    60:(* get P171 index 0 *)
        fbTD20Transaction.i_wPKE := 16#6000 OR 171;
        fbTD20Transaction.i_bIND := 0;
        fbTD20Transaction.i_dwPWE := 0;
        fbTD20Transaction.i_xExecute := TRUE;
        IF fbTD20Transaction.q_xError THEN
            iCatch := iCatch +1;
            a_TransactionErrorMesg();
            iStep := 9000;
        ELSIF fbTD20Transaction.q_xDone THEN
            fbTD20Transaction.i_xExecute := FALSE;
            IF fbTD20Transaction.q_wPKE = (16#4000 OR 171) THEN
                q_stStatus.wErrorCode_P171 := DWORD_TO_WORD(fbTD20Transaction.q_dwPWE);
                iStep := 8000;
            ELSE
                a_DriverErrorMesg();
                iStep := 9100;
            END_IF
        END_IF

    8000: (* done *)
        q_xDone := TRUE;
        IF  i_xExecute = FALSE THEN
            q_xDone:= FALSE;
            iStep := 0;
        END_IF

    9000: (* Transaction Error *)
        q_xError := TRUE;

    9100: (* Driver Error *)
        q_xError := TRUE;

END_CASE

fbTD20Transaction(
    i_wControlWord:= i_wControlWord,
    i_tTimeOut:= i_tTimeOut,
    iq_stSerialRXBuffer:= iq_stSerialRXBuffer,
    iq_stSerialTXBuffer:= iq_stSerialTXBuffer,
    q_wStatusWord=> q_stStatus.wStatusWord,
    q_wFrequency_P3=>  q_stStatus.wFrequency_P3,
    q_wVoltage_P4=> q_stStatus.wVoltage_P4,
    q_wMotorCurrent_P5=> q_stStatus.wMotorCurrent_P5,
    q_wConverterTemp_P11=> q_stStatus.wConverterTemp_P11,
    q_wPumpTemp_P127=> q_stStatus.wPumpTemp_P127);

IF fbTD20Transaction.q_xError THEN
    a_ClearStatus();
END_IF

q_abLastSentArray := fbTD20Transaction.q_abLastSentArray;
q_abLastReceivedArray := fbTD20Transaction.q_abLastReceivedArray;

ACTION a_ClearStatus:
q_stStatus.wStatusWord := 0;
q_stStatus.wFrequency_P3 := 0;
q_stStatus.wVoltage_P4 := 0;
q_stStatus.wMotorCurrent_P5 := 0;
q_stStatus.wConverterTemp_P11 := 0;
q_stStatus.wCriticalFreq_P20 := 0;
q_stStatus.wMaxCurrentFactor_P21 := 0;
q_stStatus.wSetpointFreq_P24 := 0;
q_stStatus.wMaxRunUpTime_P32 := 0;
q_stStatus.wPumpTemp_P127 := 0;
q_stStatus.wErrorCode_P171 := 0;
END_ACTION

ACTION a_DriverErrorMesg:
fbFormatString( sformat:=sDriverErrMesg,
    arg1:=F_INT(iStep),
    arg2:=F_WORD(fbTD20Transaction.q_wPKE),
    sOut => q_sResult);

a_ClearStatus();
END_ACTION

ACTION a_TransactionErrorMesg:
fbFormatString( sformat:=sTransactionErrMesg,
    arg1:=F_INT(iStep),
    arg2:=F_STRING(fbTD20Transaction.q_sResult),
    sOut => q_sResult);

a_ClearStatus();
q_xTimeout := fbTD20Transaction.q_xTimeout;
END_ACTION

END_FUNCTION_BLOCK

// ---- POUs/Serial drivers/Pumps/Oerlikon TD20/FB_TD20Transaction.TcPOU
FUNCTION_BLOCK FB_TD20Transaction
VAR_INPUT
    /// rising edge execute
    i_xExecute: BOOL;
    /// RS-485 Addrress of Pump, 0 if RS-232
    i_bAddress: BYTE;
    /// PKE Parameter number and type of access
    i_wPKE: WORD;
    /// IND Parameter index
    i_bIND: BYTE;
    /// PWE Parameter value
    i_dwPWE: DWORD;
    /// Control Word
    i_wControlWord: WORD;
    /// Maximum wait time for reply
    i_tTimeOut: TIME := TIME#1s0ms;
END_VAR
VAR_OUTPUT
    q_xDone: BOOL;
    q_xError: BOOL;
    q_xTimeout: BOOL;
    q_sResult: STRING(MAX_STRING_LENGTH);
    /// Sent data
    q_abSendData: ARRAY[0..23] OF BYTE;
    /// Received Data data
    q_abResponseData: ARRAY[0..23] OF BYTE;
    /// Received PKE
    q_wPKE: WORD;
    /// Received PWE
    q_dwPWE: DWORD;
    /// Received Status Word
    q_wStatusWord: WORD;
    /// Current stator frequency
    q_wFrequency_P3: WORD;
    /// Current intermediate circuit voltage
    q_wVoltage_P4: WORD;
    /// Current motor current
    q_wMotorCurrent_P5: WORD;
    /// Current frequency converter temperature
    q_wConverterTemp_P11: WORD;
    /// Current pump temperature
    q_wPumpTemp_P127: WORD;
    /// Last Byte Sequence Sent to Serial Device - for debugging
    q_abLastSentArray: ARRAY[0..23] OF BYTE;
    /// Last Byte Sequence Received from Serial Device - for debugging
    q_abLastReceivedArray: ARRAY[0..23] OF BYTE;
END_VAR
VAR_IN_OUT
    iq_stSerialRXBuffer: ComBuffer;
    iq_stSerialTXBuffer: ComBuffer;
END_VAR
VAR
    rtExecute: R_TRIG;
    iStep: INT;
    fbClearComBuffer: ClearComBuffer;
    tonTimeout: TON;
    wTemp: WORD;
    dwTemp: DWORD;
    i: INT;
    fbSendData: SendData;
    fbReceiveData: ReceiveData;
    bRXChecksum: BYTE;
    bRXAddress: BYTE;
    nPrefix : BYTE := 16#02;
END_VAR

(* This function block performs serial transactions with an Oerlikon TD20 *)

(* rising edge trigger *)
rtExecute(CLK:= i_xExecute);
IF rtExecute.Q THEN
    q_xDone	:= FALSE;
    q_xError := FALSE;
    q_xTimeout := FALSE;
    q_sResult:= '';
    MEMSET(destAddr:=ADR(q_abSendData), fillByte:=0, n:=SIZEOF(q_abSendData));
    MEMSET(destAddr:=ADR(q_abResponseData), fillByte:=0, n:=SIZEOF(q_abResponseData));
    iStep := 10;
END_IF

CASE iStep OF
    0:
        ; (* idle *)

    10: (* clear com buffers *)
        fbClearComBuffer(Buffer:= iq_stSerialRXBuffer);
        fbClearComBuffer(Buffer:= iq_stSerialTXBuffer);

        (* build the send data *)
        (* byte 0 STX *)
        q_abSendData[0] := 2; (* STX *)

        (* byte 1 LGE - Length *)
        q_abSendData[1] := 22;

        (* byte 2 ADR - Address for RS-485, use 0 for RS-232 *)
        q_abSendData[2] := i_bAddress;

        (* bytes 3-4 PKE - Parameter Number and Type of Access *)
        wTemp :=  HOST_TO_BE16(i_wPKE);
        MEMCPY(destAddr:= ADR(q_abSendData[3]), srcAddr:=ADR(wTemp), n:=2);

        (* byte 5 is reserved *)
        (* byte 6 IND - Parameter index *)
        q_abSendData[6] := i_bIND;

        (* bytes 7-10 - Parameter Value *)
        dwTemp := HOST_TO_BE32(i_dwPWE);
        MEMCPY(destAddr:= ADR(q_abSendData[7]), srcAddr:=ADR(dwTemp), n:=4);

        (* bytes 11-12 - control word *)
        wTemp :=  HOST_TO_BE16(i_wControlWord);
        MEMCPY(destAddr:= ADR(q_abSendData[11]), srcAddr:=ADR(wTemp), n:=2);

        (* rest of the bytes for any read or write are 0 *)
        (* generate checksum *)
        q_abSendData[23] := F_CalcTD20Checksum(i_abData:=q_abSendData);

        (* send the data *)
        fbSendData(
            pSendData:= ADR(q_abSendData),
            Length:= 24,
            TXbuffer:= iq_stSerialTXBuffer);


        q_abLastSentArray := q_abSendData;
        iStep := iStep + 10;

    20: (* Finish sending the data *)
        IF fbSendData.Busy THEN
            fbSendData( TXbuffer:= iq_stSerialTXBuffer );
        ELSIF fbSendData.Error <> 0 THEN
            q_sResult := CONCAT('In step 20 fbSendData resulted in error: ', INT_TO_STRING(fbSendData.Error));
            iStep := 9000;
        ELSIF NOT fbSendData.Busy THEN
            iStep := iStep + 10;
        END_IF
        (* Reset receive *)
        fbReceiveData(
            pReceiveData:= ADR(q_abResponseData),
            Reset:= TRUE,
            RXbuffer:= iq_stSerialRXBuffer);
        tonTimeout(IN:= FALSE);

    30: (* Get reply *)
        fbReceiveData(
            pReceiveData:= ADR(q_abResponseData),
            SizeReceiveData:= 24,
            Timeout:= i_tTimeOut,
            Reset:= FALSE,
            RXbuffer:= iq_stSerialRXBuffer,
            pPrefix := ADR(nPrefix), LenPrefix:=1 );
        tonTimeout(IN:= TRUE, PT:= i_tTimeOut);
        IF fbReceiveData.Error <> 0 THEN
            q_sResult := CONCAT('In step 30 fbReceiveData resulted in error: ', INT_TO_STRING(fbReceiveData.Error));
            iStep := 9000;
        ELSIF fbReceiveData.RxTimeout OR tonTimeout.Q THEN
            q_sResult := 'Device failed to reply within timeout period';
            q_xTimeout := TRUE;
            iStep := 9000;
        ELSIF fbReceiveData.DataReceived THEN
            q_abLastReceivedArray := q_abResponseData;
            bRXChecksum := F_CalcTD20Checksum(q_abResponseData);
            bRXAddress := q_abResponseData[2];
            MEMCPY(destAddr:=ADR(wTemp) , srcAddr:=ADR(q_abResponseData[3]), n:=2);
            q_wPKE := BE16_TO_HOST(wTemp);
            MEMCPY(destAddr:=ADR(dwTemp) , srcAddr:=ADR(q_abResponseData[7]), n:=4);
            q_dwPWE := BE32_TO_HOST(dwTemp);

            IF bRXChecksum <> q_abResponseData[23] THEN
                q_sResult := 'Invalid checksum on received data.';
                iStep := 9000;
            ELSIF i_bAddress <> bRXAddress THEN
                q_sResult := 'Invalid unit address on received data.';
                iStep := 9000;
            ELSIF (q_wPKE AND 16#F000) = 2#0111000000000000 THEN
                q_sResult := 'Frequency converter cannot run the command.';
                iStep := 9000;
            ELSIF (Q_wPKE AND 16#F000) = 2#1000000000000000 THEN
                q_sResult := 'During write access: no permission to write.';
                iStep := 9000;
            ELSE
                MEMCPY(destAddr:=ADR(wTemp) , srcAddr:=ADR(q_abResponseData[11]), n:=2);
                q_wStatusWord := BE16_TO_HOST(wTemp);
                MEMCPY(destAddr:=ADR(wTemp) , srcAddr:=ADR(q_abResponseData[13]), n:=2);
                q_wFrequency_P3:= BE16_TO_HOST(wTemp);
                MEMCPY(destAddr:=ADR(wTemp) , srcAddr:=ADR(q_abResponseData[21]), n:=2);
                q_wVoltage_P4:= BE16_TO_HOST(wTemp);
                MEMCPY(destAddr:=ADR(wTemp) , srcAddr:=ADR(q_abResponseData[17]), n:=2);
                q_wMotorCurrent_P5:= BE16_TO_HOST(wTemp);
                MEMCPY(destAddr:=ADR(wTemp) , srcAddr:=ADR(q_abResponseData[15]), n:=2);
                q_wConverterTemp_P11:= BE16_TO_HOST(wTemp);
                MEMCPY(destAddr:=ADR(wTemp) , srcAddr:=ADR(q_abResponseData[19]), n:=2);
                q_wPumpTemp_P127:= BE16_TO_HOST(wTemp);
                q_sResult := 'Success.';
                q_xDone:= TRUE;
                iStep := 100;
            END_IF
        END_IF

    100: (* done *)
        IF  i_xExecute = FALSE THEN
            q_xDone:= FALSE;
            iStep := 0;
        END_IF

    9000:
        q_wPKE:= 0;
        q_dwPWE:= 0;
        q_wStatusWord:= 0;
        q_wFrequency_P3:= 0;
        q_wVoltage_P4:= 0;
        q_wMotorCurrent_P5:= 0;
        q_wConverterTemp_P11:= 0;
        q_wPumpTemp_P127:= 0;
        q_xError := TRUE;;




END_CASE

END_FUNCTION_BLOCK

// ---- POUs/Serial drivers/Pumps/Oerlikon TD20/F_CalcTD20Checksum.TcPOU
FUNCTION F_CalcTD20Checksum : BYTE
VAR_INPUT
    i_abData: ARRAY[0..23] OF BYTE;
END_VAR
VAR
    bChecksum: BYTE;
    i: INT;
END_VAR

bChecksum := i_abData[0];
FOR i:=1 TO 22 DO
    bChecksum := bChecksum XOR i_abData[i];
END_FOR
F_CalcTD20Checksum := bChecksum;

END_FUNCTION

// ---- POUs/Serial drivers/Pumps/Oerlikon TD20/FB_OERLIKON_TO_PTM.TcPOU
FUNCTION_BLOCK FB_OERLIKON_TO_PTM
VAR_IN_OUT
    iq_stPTM: ST_LeyboldPTM;
    iq_stOerlikon_stat: ST_TD20Status;
END_VAR

(* This function block is used to map the IO points from the Oerlikon structures
to the generic turbo structures *)

(* Readbacks *)
iq_stPTM.i_xAccel := iq_stOerlikon_stat.wStatusWord.4;
iq_stPTM.i_xDecel := iq_stOerlikon_stat.wStatusWord.5;
iq_stPTM.i_xAtSpd := iq_stOerlikon_stat.wStatusWord.10;
iq_stPTM.q_xRemote := iq_stOerlikon_stat.wStatusWord.15; (* Remote control enabled *)
iq_stPTM.i_diCurSpd := WORD_TO_DINT(iq_stOerlikon_stat.wFrequency_P3);
iq_stPTM.i_diPwr := LREAL_TO_DINT(WORD_TO_DINT(iq_stOerlikon_stat.wMotorCurrent_P5 * iq_stOerlikon_stat.wVoltage_P4)*0.01); (*Current in units 0.1 A and voltage in units 0.1V, TD20 manual page 23*)
iq_stPTM.i_diElecTemp := WORD_TO_DINT(iq_stOerlikon_stat.wConverterTemp_P11);
//iq_stPTM.i_diPumpTemp := WORD_TO_DINT(iq_stOerlikon_stat.wPumpTemp_P127);

(* Faults and warnings *)
//iq_stPTM.xFault := iq_stOerlikon_stat.wStatusWord.3;
iq_stPTM.i_xTempFault := iq_stOerlikon_stat.wStatusWord.7; (* specified as a temperature warning but it could be a fault *)
//iq_stPTM.xWarn := iq_stOerlikon_stat.wStatusWord.14; (* warning summary bit *)

END_FUNCTION_BLOCK

// ---- POUs/Serial drivers/Pumps/Oerlikon TD400/FB_OERLIKON_TD400_COM.TcPOU
FUNCTION_BLOCK FB_OERLIKON_TD400_COM
VAR_INPUT
END_VAR
VAR
    tTimeOut : TIME := TIME#1S0MS;
    fbTD400SerialDriver : FB_TD400SerialDriver;
END_VAR
VAR_IN_OUT
    SerialRXBuffer : ComBuffer;
    SerialTXBuffer : ComBuffer;
    stTD400Control : ST_TD400Control;
END_VAR
VAR_OUTPUT
    stTD400Status : ST_TD400Status;
END_VAR

(* This program is called from Serial PTM IO *)

(* scan the pumps one at a time *)//MG???
fbTD400SerialDriver(
    i_xExecute:= TRUE,
    i_tTimeOut:= tTimeOut,
    i_wControlWord:= 16#0000,
    iq_stControl:= stTD400Control,
    iq_stSerialRXBuffer:= SerialRXBuffer,
    iq_stSerialTXBuffer:= SerialTXBuffer,
    q_xDone=> ,
    q_xError=> ,
    q_xTimeout=> ,
    q_sResult=> ,
    q_stStatus=> stTD400Status);

IF fbTD400SerialDriver.q_xDone
    OR fbTD400SerialDriver.q_xError
    OR fbTD400SerialDriver.q_xTimeout THEN
        (* reset for next time *)
        fbTD400SerialDriver(i_xExecute:= FALSE, iq_stSerialRXBuffer:= SerialRXBuffer, iq_stSerialTXBuffer:= SerialTXBuffer, iq_stControl:= stTD400Control);
END_IF

END_FUNCTION_BLOCK

// ---- POUs/Serial drivers/Pumps/Oerlikon TD400/FB_TD400SerialDriver.TcPOU
FUNCTION_BLOCK FB_TD400SerialDriver
VAR_INPUT
    /// rising edge execute
    i_xExecute: BOOL;
    /// Maximum wait time for reply
    i_tTimeOut: TIME := TIME#1s0ms;
    i_wControlWord: WORD;
END_VAR
VAR_OUTPUT
    q_xDone: BOOL;
    q_xError: BOOL;
    q_xTimeout: BOOL;
    q_sResult: STRING(255);
    q_stStatus: ST_TD400Status;
    /// Last Byte Sequence Sent to Serial Device - for debugging
    q_abLastSentArray: ARRAY[0..23] OF BYTE;
    /// Last Byte Sequence Received from Serial Device - for debugging
    q_abLastReceivedArray: ARRAY[0..23] OF BYTE;
END_VAR
VAR_IN_OUT
    iq_stSerialRXBuffer: ComBuffer;
    iq_stSerialTXBuffer: ComBuffer;
    iq_stControl: ST_TD400Control;
END_VAR
VAR
    rtExecute: R_TRIG;
    rtTransDone: R_TRIG;
    iStep: INT;
    fbTD400Transaction: FB_TD400Transaction;
    fbFormatString: FB_FormatString;
    iCatch: INT;
    sTransactionErrMesg : STRING := 'In step %d fbTD20Transaction failed with message: %s';
    sDriverErrMesg		: STRING := 'In step %d FB_TD20SerialDriver failed with unexpected PKE reply: %X';
    bSetFreq : BOOL := FALSE; //flag to write to controller to set new frequency
    nOldSetSetpointFreq_P24 : WORD; //local value for setpoint frequency parameter to compare with new value
    bControlDisabled : BOOL := TRUE; //flag to enable setting frequency
END_VAR

(* This function block performs serial transactions with a Oerlikon TD400 Pump controller *)
//Wait until all needed parameters received to enable control to set frequency
IF q_stStatus.wMinSetpointFreq_P19 <> 0 AND q_stStatus.wMaxSetpointFreq_P18 <> 0 AND q_stStatus.wSetpointFreq_P24 <> 0 THEN
    //On first pass update Set frequency parameter with value from controller
    IF bControlDisabled THEN
        iq_stControl.wSetSetpointFreq_P24 := q_stStatus.wSetpointFreq_P24;
        nOldSetSetpointFreq_P24 := q_stStatus.wSetpointFreq_P24;
        bControlDisabled := FALSE;
        bSetFreq := FALSE;
    ELSE
        IF nOldSetSetpointFreq_P24 <> iq_stControl.wSetSetpointFreq_P24 THEN
            nOldSetSetpointFreq_P24 := iq_stControl.wSetSetpointFreq_P24;
            bSetFreq := TRUE;
        END_IF
    END_IF
ELSE
    iq_stControl.wSetSetpointFreq_P24 := q_stStatus.wSetpointFreq_P24;
    bControlDisabled := TRUE;
    bSetFreq := FALSE;
END_IF

(* rising edge trigger *)
rtExecute(CLK:= i_xExecute);
IF rtExecute.Q  THEN
    q_xDone	:= FALSE;
    q_xError := FALSE;
    q_xTimeout := FALSE;
    q_sResult:= '';
    iStep := 10;
END_IF

CASE iStep OF
    0: (* idle *)
        ;

    10: (* assure rising edge *)
        fbTD400Transaction.i_xExecute := FALSE;
        iStep := iStep + 10;

    20:(* get P20 *)
        fbTD400Transaction.i_wPKE := 16#1000 OR 20;
        fbTD400Transaction.i_bIND := 0;
        fbTD400Transaction.i_dwPWE := 0;
        fbTD400Transaction.i_xExecute := TRUE;

        IF fbTD400Transaction.q_xError THEN
            iCatch := iCatch +1;
            a_TransactionErrorMesg();
            iStep := 9000;
        ELSIF fbTD400Transaction.q_xDone THEN
            fbTD400Transaction.i_xExecute := FALSE;
            IF fbTD400Transaction.q_wPKE = (16#1000 OR 20) THEN
                q_stStatus.wCriticalFreq_P20 := DWORD_TO_WORD(fbTD400Transaction.q_dwPWE);
                iStep := iStep + 10;
            ELSE
                a_DriverErrorMesg();
                iStep := 9100;
            END_IF
        END_IF

    30:(* set P24 *)
        IF bSetFreq THEN
            fbTD400Transaction.i_wPKE := 16#2000 OR 24;
            fbTD400Transaction.i_bIND := 0;
            fbTD400Transaction.i_dwPWE := WORD_TO_DWORD(iq_stControl.wSetSetpointFreq_P24);
            fbTD400Transaction.i_xExecute := TRUE;

            IF fbTD400Transaction.q_xError THEN
                iCatch := iCatch +1;
                a_TransactionErrorMesg();
                iStep := 9000;
                bSetFreq := FALSE;
            ELSIF fbTD400Transaction.q_xDone THEN
                fbTD400Transaction.i_xExecute := FALSE;
                bSetFreq := FALSE;
                IF fbTD400Transaction.q_wPKE = (16#1000 OR 24) THEN
                    q_stStatus.wSetpointFreq_P24 := DWORD_TO_WORD(fbTD400Transaction.q_dwPWE);
                    iStep := iStep + 10;
                ELSE
                    a_DriverErrorMesg();
                    iStep := 9100;
                END_IF
            END_IF
        ELSE
            iStep := iStep + 10;
        END_IF

    40:(* get P24 *)
        fbTD400Transaction.i_wPKE := 16#1000 OR 24;
        fbTD400Transaction.i_bIND := 0;
        fbTD400Transaction.i_dwPWE := 0;
        fbTD400Transaction.i_xExecute := TRUE;
        IF fbTD400Transaction.q_xError THEN
            iCatch := iCatch +1;
            a_TransactionErrorMesg();
            iStep := 9000;
        ELSIF fbTD400Transaction.q_xDone THEN
            fbTD400Transaction.i_xExecute := FALSE;
            IF fbTD400Transaction.q_wPKE = (16#1000 OR 24) THEN
                q_stStatus.wSetpointFreq_P24 := DWORD_TO_WORD(fbTD400Transaction.q_dwPWE);
                iStep := iStep + 10;
            ELSE
                a_DriverErrorMesg();
                iStep := 9100;
            END_IF
        END_IF

    50:(* get P32 *)
        fbTD400Transaction.i_wPKE := 16#1000 OR 32;
        fbTD400Transaction.i_bIND := 0;
        fbTD400Transaction.i_dwPWE := 0;
        fbTD400Transaction.i_xExecute := TRUE;
        IF fbTD400Transaction.q_xError THEN
            iCatch := iCatch +1;
            a_TransactionErrorMesg();
            iStep := 9000;
        ELSIF fbTD400Transaction.q_xDone THEN
            fbTD400Transaction.i_xExecute := FALSE;
            IF fbTD400Transaction.q_wPKE = (16#1000 OR 32) THEN
                q_stStatus.wMaxRunUpTime_P32 := DWORD_TO_WORD(fbTD400Transaction.q_dwPWE);
                iStep := iStep + 10;
            ELSE
                a_DriverErrorMesg();
                iStep := 9100;
            END_IF
        END_IF

    60:(* get P171 index 0 *)
        fbTD400Transaction.i_wPKE := 16#6000 OR 171;
        fbTD400Transaction.i_bIND := 0;
        fbTD400Transaction.i_dwPWE := 0;
        fbTD400Transaction.i_xExecute := TRUE;
        IF fbTD400Transaction.q_xError THEN
            iCatch := iCatch +1;
            a_TransactionErrorMesg();
            iStep := 9000;
        ELSIF fbTD400Transaction.q_xDone THEN
            fbTD400Transaction.i_xExecute := FALSE;
            IF fbTD400Transaction.q_wPKE = (16#4000 OR 171) THEN
                q_stStatus.wErrorCode_P171 := DWORD_TO_WORD(fbTD400Transaction.q_dwPWE);
                //iStep := 8000;
                iStep := iStep + 10;
            ELSE
                a_DriverErrorMesg();
                iStep := 9100;
            END_IF
        END_IF

    70:(* get P18 *)
        fbTD400Transaction.i_wPKE := 16#1000 OR 18;
        fbTD400Transaction.i_bIND := 0;
        fbTD400Transaction.i_dwPWE := 0;
        fbTD400Transaction.i_xExecute := TRUE;
        IF fbTD400Transaction.q_xError THEN
            iCatch := iCatch +1;
            a_TransactionErrorMesg();
            iStep := 9000;
        ELSIF fbTD400Transaction.q_xDone THEN
            fbTD400Transaction.i_xExecute := FALSE;
            IF fbTD400Transaction.q_wPKE = (16#1000 OR 18) THEN
                q_stStatus.wMaxSetpointFreq_P18 := DWORD_TO_WORD(fbTD400Transaction.q_dwPWE);
                iStep := iStep + 10;
            ELSE
                a_DriverErrorMesg();
                iStep := 9100;
            END_IF
        END_IF

    80:(* get P19 *)
        fbTD400Transaction.i_wPKE := 16#1000 OR 19;
        fbTD400Transaction.i_bIND := 0;
        fbTD400Transaction.i_dwPWE := 0;
        fbTD400Transaction.i_xExecute := TRUE;
        IF fbTD400Transaction.q_xError THEN
            iCatch := iCatch +1;
            a_TransactionErrorMesg();
            iStep := 9000;
        ELSIF fbTD400Transaction.q_xDone THEN
            fbTD400Transaction.i_xExecute := FALSE;
            IF fbTD400Transaction.q_wPKE = (16#1000 OR 19) THEN
                q_stStatus.wMinSetpointFreq_P19 := DWORD_TO_WORD(fbTD400Transaction.q_dwPWE);
                iStep := 8000;
            ELSE
                a_DriverErrorMesg();
                iStep := 9100;
            END_IF
        END_IF

    8000: (* done *)
        q_xDone := TRUE;
        IF  i_xExecute = FALSE THEN
            q_xDone:= FALSE;
            iStep := 0;
        END_IF

    9000: (* Transaction Error *)
        q_xError := TRUE;

    9100: (* Driver Error *)
        q_xError := TRUE;

END_CASE

fbTD400Transaction(
    i_wControlWord:= i_wControlWord,
    i_tTimeOut:= i_tTimeOut,
    iq_stSerialRXBuffer:= iq_stSerialRXBuffer,
    iq_stSerialTXBuffer:= iq_stSerialTXBuffer,
    q_wStatusWord=> q_stStatus.wStatusWord,
    q_wFrequency_P3=>  q_stStatus.wFrequency_P3,
    q_wVoltage_P4=> q_stStatus.wVoltage_P4,
    q_wMotorCurrent_P5=> q_stStatus.wMotorCurrent_P5,
    q_wConverterTemp_P11=> q_stStatus.wConverterTemp_P11,
    q_wPumpTemp_P127=> q_stStatus.wPumpTemp_P127);

IF fbTD400Transaction.q_xError THEN
    a_ClearStatus();
END_IF

q_abLastSentArray := fbTD400Transaction.q_abLastSentArray;
q_abLastReceivedArray := fbTD400Transaction.q_abLastReceivedArray;

ACTION a_ClearStatus:
q_stStatus.wStatusWord := 0;
q_stStatus.wFrequency_P3 := 0;
q_stStatus.wVoltage_P4 := 0;
q_stStatus.wMotorCurrent_P5 := 0;
q_stStatus.wConverterTemp_P11 := 0;
q_stStatus.wMaxSetpointFreq_P18 := 0;
q_stStatus.wMinSetpointFreq_P19 := 0;
q_stStatus.wCriticalFreq_P20 := 0;
//q_stStatus.wMaxCurrentFactor_P21 := 0;
q_stStatus.wSetpointFreq_P24 := 0;
q_stStatus.wMaxRunUpTime_P32 := 0;
q_stStatus.wPumpTemp_P127 := 0;
q_stStatus.wErrorCode_P171 := 0;
END_ACTION

ACTION a_DriverErrorMesg:
fbFormatString( sformat:=sDriverErrMesg,
    arg1:=F_INT(iStep),
    arg2:=F_WORD(fbTD400Transaction.q_wPKE),
    sOut => q_sResult);

a_ClearStatus();
END_ACTION

ACTION a_TransactionErrorMesg:
fbFormatString( sformat:=sTransactionErrMesg,
    arg1:=F_INT(iStep),
    arg2:=F_STRING(fbTD400Transaction.q_sResult),
    sOut => q_sResult);

a_ClearStatus();
q_xTimeout := fbTD400Transaction.q_xTimeout;
END_ACTION

END_FUNCTION_BLOCK

// ---- POUs/Serial drivers/Pumps/Oerlikon TD400/FB_TD400Transaction.TcPOU
FUNCTION_BLOCK FB_TD400Transaction
VAR_INPUT
    /// rising edge execute
    i_xExecute: BOOL;
    /// RS-485 Addrress of Pump, 0 if RS-232
    i_bAddress: BYTE;
    /// PKE Parameter number and type of access
    i_wPKE: WORD;
    /// IND Parameter index
    i_bIND: BYTE;
    /// PWE Parameter value
    i_dwPWE: DWORD;
    /// Control Word
    i_wControlWord: WORD;
    /// Maximum wait time for reply
    i_tTimeOut: TIME := TIME#1s0ms;
END_VAR
VAR_OUTPUT
    q_xDone: BOOL;
    q_xError: BOOL;
    q_xTimeout: BOOL;
    q_sResult: STRING(MAX_STRING_LENGTH);
    /// Sent data
    q_abSendData: ARRAY[0..23] OF BYTE;
    /// Received Data data
    q_abResponseData: ARRAY[0..23] OF BYTE;
    /// Received PKE
    q_wPKE: WORD;
    /// Received PWE
    q_dwPWE: DWORD;
    /// Received Status Word
    q_wStatusWord: WORD;
    /// Current stator frequency
    q_wFrequency_P3: WORD;
    /// Current intermediate circuit voltage
    q_wVoltage_P4: WORD;
    /// Current motor current
    q_wMotorCurrent_P5: WORD;
    /// Current frequency converter temperature
    q_wConverterTemp_P11: WORD;
    /// Current pump temperature
    q_wPumpTemp_P127: WORD;
    /// Last Byte Sequence Sent to Serial Device - for debugging
    q_abLastSentArray: ARRAY[0..23] OF BYTE;
    /// Last Byte Sequence Received from Serial Device - for debugging
    q_abLastReceivedArray: ARRAY[0..23] OF BYTE;
END_VAR
VAR_IN_OUT
    iq_stSerialRXBuffer: ComBuffer;
    iq_stSerialTXBuffer: ComBuffer;
END_VAR
VAR
    rtExecute: R_TRIG;
    iStep: INT;
    fbClearComBuffer: ClearComBuffer;
    tonTimeout: TON;
    wTemp: WORD;
    dwTemp: DWORD;
    i: INT;
    fbSendData: SendData;
    fbReceiveData: ReceiveData;
    bRXChecksum: BYTE;
    bRXAddress: BYTE;
    nPrefix : BYTE := 16#02;
END_VAR

(* This function block performs serial transactions with an Oerlikon TD20 *)

(* rising edge trigger *)
rtExecute(CLK:= i_xExecute);
IF rtExecute.Q THEN
    q_xDone	:= FALSE;
    q_xError := FALSE;
    q_xTimeout := FALSE;
    q_sResult:= '';
    MEMSET(destAddr:=ADR(q_abSendData), fillByte:=0, n:=SIZEOF(q_abSendData));
    MEMSET(destAddr:=ADR(q_abResponseData), fillByte:=0, n:=SIZEOF(q_abResponseData));
    iStep := 10;
END_IF

CASE iStep OF
    0:
        ; (* idle *)

    10: (* clear com buffers *)
        fbClearComBuffer(Buffer:= iq_stSerialRXBuffer);
        fbClearComBuffer(Buffer:= iq_stSerialTXBuffer);

        (* build the send data *)
        (* byte 0 STX *)
        q_abSendData[0] := 2; (* STX *)

        (* byte 1 LGE - Length *)
        q_abSendData[1] := 22;

        (* byte 2 ADR - Address for RS-485, use 0 for RS-232 *)
        q_abSendData[2] := i_bAddress;

        (* bytes 3-4 PKE - Parameter Number and Type of Access *)
        wTemp :=  HOST_TO_BE16(i_wPKE);
        MEMCPY(destAddr:= ADR(q_abSendData[3]), srcAddr:=ADR(wTemp), n:=2);

        (* byte 5 is reserved *)
        (* byte 6 IND - Parameter index *)
        q_abSendData[6] := i_bIND;

        (* bytes 7-10 - Parameter Value *)
        dwTemp := HOST_TO_BE32(i_dwPWE);
        MEMCPY(destAddr:= ADR(q_abSendData[7]), srcAddr:=ADR(dwTemp), n:=4);

        (* bytes 11-12 - control word *)
        wTemp :=  HOST_TO_BE16(i_wControlWord);
        MEMCPY(destAddr:= ADR(q_abSendData[11]), srcAddr:=ADR(wTemp), n:=2);

        (* rest of the bytes for any read or write are 0 *)
        (* generate checksum *)
        q_abSendData[23] := F_CalcTD20Checksum(i_abData:=q_abSendData);

        (* send the data *)
        fbSendData(
            pSendData:= ADR(q_abSendData),
            Length:= 24,
            TXbuffer:= iq_stSerialTXBuffer);


        q_abLastSentArray := q_abSendData;
        iStep := iStep + 10;

    20: (* Finish sending the data *)
        IF fbSendData.Busy THEN
            fbSendData( TXbuffer:= iq_stSerialTXBuffer );
        ELSIF fbSendData.Error <> 0 THEN
            q_sResult := CONCAT('In step 20 fbSendData resulted in error: ', INT_TO_STRING(fbSendData.Error));
            iStep := 9000;
        ELSIF NOT fbSendData.Busy THEN
            iStep := iStep + 10;
        END_IF
        (* Reset receive *)
        fbReceiveData(
            pReceiveData:= ADR(q_abResponseData),
            Reset:= TRUE,
            RXbuffer:= iq_stSerialRXBuffer);
        tonTimeout(IN:= FALSE);

    30: (* Get reply *)
        fbReceiveData(
            pReceiveData:= ADR(q_abResponseData),
            SizeReceiveData:= 24,
            Timeout:= i_tTimeOut,
            Reset:= FALSE,
            RXbuffer:= iq_stSerialRXBuffer,
            pPrefix := ADR(nPrefix), LenPrefix:=1 );
        tonTimeout(IN:= TRUE, PT:= i_tTimeOut);
        IF fbReceiveData.Error <> 0 THEN
            q_sResult := CONCAT('In step 30 fbReceiveData resulted in error: ', INT_TO_STRING(fbReceiveData.Error));
            iStep := 9000;
        ELSIF fbReceiveData.RxTimeout OR tonTimeout.Q THEN
            q_sResult := 'Device failed to reply within timeout period';
            q_xTimeout := TRUE;
            iStep := 9000;
        ELSIF fbReceiveData.DataReceived THEN
            q_abLastReceivedArray := q_abResponseData;
            bRXChecksum := F_CalcTD400Checksum(q_abResponseData);
            bRXAddress := q_abResponseData[2];
            MEMCPY(destAddr:=ADR(wTemp) , srcAddr:=ADR(q_abResponseData[3]), n:=2);
            q_wPKE := BE16_TO_HOST(wTemp);
            MEMCPY(destAddr:=ADR(dwTemp) , srcAddr:=ADR(q_abResponseData[7]), n:=4);
            q_dwPWE := BE32_TO_HOST(dwTemp);

            IF bRXChecksum <> q_abResponseData[23] THEN
                q_sResult := 'Invalid checksum on received data.';
                iStep := 9000;
            ELSIF i_bAddress <> bRXAddress THEN
                q_sResult := 'Invalid unit address on received data.';
                iStep := 9000;
            ELSIF (q_wPKE AND 16#F000) = 2#0111000000000000 THEN
                q_sResult := 'Frequency converter cannot run the command.';
                iStep := 9000;
            ELSIF (Q_wPKE AND 16#F000) = 2#1000000000000000 THEN
                q_sResult := 'During write access: no permission to write.';
                iStep := 9000;
            ELSE
                MEMCPY(destAddr:=ADR(wTemp) , srcAddr:=ADR(q_abResponseData[11]), n:=2);
                q_wStatusWord := BE16_TO_HOST(wTemp);
                MEMCPY(destAddr:=ADR(wTemp) , srcAddr:=ADR(q_abResponseData[13]), n:=2);
                q_wFrequency_P3:= BE16_TO_HOST(wTemp);
                MEMCPY(destAddr:=ADR(wTemp) , srcAddr:=ADR(q_abResponseData[21]), n:=2);
                q_wVoltage_P4:= BE16_TO_HOST(wTemp);
                MEMCPY(destAddr:=ADR(wTemp) , srcAddr:=ADR(q_abResponseData[17]), n:=2);
                q_wMotorCurrent_P5:= BE16_TO_HOST(wTemp);
                MEMCPY(destAddr:=ADR(wTemp) , srcAddr:=ADR(q_abResponseData[15]), n:=2);
                q_wConverterTemp_P11:= BE16_TO_HOST(wTemp);
                MEMCPY(destAddr:=ADR(wTemp) , srcAddr:=ADR(q_abResponseData[19]), n:=2);
                q_wPumpTemp_P127:= BE16_TO_HOST(wTemp);
                q_sResult := 'Success.';
                q_xDone:= TRUE;
                iStep := 100;
            END_IF
        END_IF

    100: (* done *)
        IF  i_xExecute = FALSE THEN
            q_xDone:= FALSE;
            iStep := 0;
        END_IF

    9000:
        q_wPKE:= 0;
        q_dwPWE:= 0;
        q_wStatusWord:= 0;
        q_wFrequency_P3:= 0;
        q_wVoltage_P4:= 0;
        q_wMotorCurrent_P5:= 0;
        q_wConverterTemp_P11:= 0;
        q_wPumpTemp_P127:= 0;
        q_xError := TRUE;

END_CASE

END_FUNCTION_BLOCK

// ---- POUs/Serial drivers/Pumps/Oerlikon TD400/F_CalcTD400Checksum.TcPOU
FUNCTION F_CalcTD400Checksum : BYTE
VAR_INPUT
    i_abData: ARRAY[0..23] OF BYTE;
END_VAR
VAR
    bChecksum: BYTE;
    i: INT;
END_VAR

bChecksum := i_abData[0];
FOR i:=1 TO 22 DO
    bChecksum := bChecksum XOR i_abData[i];
END_FOR
F_CalcTD400Checksum := bChecksum;

END_FUNCTION

// ---- POUs/Serial drivers/Pumps/Oerlikon TD400/FB_OERLIKON_TD400_TO_PTM.TcPOU
FUNCTION_BLOCK FB_OERLIKON_TD400_TO_PTM
VAR_IN_OUT
    iq_stPTM : ST_LeyboldPTM;
    iq_stTD400Status : ST_TD400Status;
    iq_stTD400Control : ST_TD400Control;
END_VAR
VAR
END_VAR

(* This function block is used to map the IO points from the Oerlikon TD400 structures
to the generic turbo structures *)
//Use this function to map IO as a temporary solution if we don't change method FB_PTM_TurboDrive.M_Serial_IO and ST_LeyboldPTM structure

(* Readbacks *)
iq_stPTM.i_xAccel := iq_stTD400Status.wStatusWord.4;
iq_stPTM.i_xDecel := iq_stTD400Status.wStatusWord.5;
//iq_stPTM.i_xAtSpd := iq_stTD400Status.wStatusWord.10;
iq_stPTM.q_xRemote := iq_stTD400Status.wStatusWord.15; (* Remote control enabled *)
iq_stPTM.i_diCurSpd := WORD_TO_DINT(iq_stTD400Status.wFrequency_P3);
iq_stPTM.i_rCurrentMon := WORD_TO_INT(iq_stTD400Status.wMotorCurrent_P5)*0.1; (*Current in units 0.1 A, TD400 Interface manual page 6*)
iq_stPTM.i_diPwr := LREAL_TO_DINT(WORD_TO_DINT(iq_stTD400Status.wMotorCurrent_P5 * iq_stTD400Status.wVoltage_P4)*0.1); (*Current in units 0.1 A, TD400 Interface manual page 6*)
iq_stPTM.i_diElecTemp := WORD_TO_DINT(iq_stTD400Status.wConverterTemp_P11);
iq_stPTM.i_rTempMon := WORD_TO_INT(iq_stTD400Status.wPumpTemp_P127);

(* Faults and warnings *)
//iq_stPTM.xFault := iq_stTD400Status.wStatusWord.3;
iq_stPTM.i_xTempFault := iq_stTD400Status.wStatusWord.7; (* specified as a temperature warning but it could be a fault *)
iq_stPTM.i_xWarn := iq_stTD400Status.wStatusWord.14; (* warning summary bit *)

(* Controls *)
iq_stTD400Control.wSetSetpointFreq_P24 := LIMIT (iq_stTD400Status.wMinSetpointFreq_P19, iq_stTD400Control.wSetSetpointFreq_P24, iq_stTD400Status.wMaxSetpointFreq_P18);

END_FUNCTION_BLOCK

// ---- POUs/Serial drivers/Pumps/Pfeiffer/FB_PfeifferSerialDriver.TcPOU
FUNCTION_BLOCK FB_PfeifferSerialDriver
VAR_INPUT
    /// rising edge execute
    i_xExecute: BOOL;
    /// Maximum wait time for reply
    i_tTimeOut: TIME := TIME#1s0ms;
    i_stControl: ST_PfeifferControl;
END_VAR
VAR_OUTPUT
    q_xDone: BOOL;
    q_xError: BOOL;
    q_xTimeout: BOOL;
    q_sResult: STRING(255);
    /// Last String Sent to Serial Device - for debugging
    q_sLastSentString: STRING;
    /// Last String Received from Serial Device - for debugging
    q_sLastReceivedString: STRING;
    q_stStatus: ST_PfeifferStatus;
END_VAR
VAR_IN_OUT
    iq_stSerialRXBuffer: ComBuffer;
    iq_stSerialTXBuffer: ComBuffer;
END_VAR
VAR
    rtExecute: R_TRIG;
    iStep: INT;
    sSendData: STRING;
    fbPfeifferTransaction: FB_PfeifferTransaction;
    fbFormatString: FB_FormatString;
    diOldSetRotationSpeed_707 :DINT;
END_VAR

(* This function block performs serial transactions with a Pfeiffer RC400 Pump controller *)

IF NOT i_stControl.xEnableComm THEN
    _A_ClearStatus();
END_IF

(* rising edge trigger *)
rtExecute(CLK:= i_xExecute);
IF rtExecute.Q  THEN
    q_xDone	:= FALSE;
    q_xError := FALSE;
    q_sResult:= '';
    IF  i_stControl.xEnableComm THEN
        a_ClearTrans();  (* to provide rising edge for execute *)
        iStep := 10;
    ELSE
        q_sResult := 'Communication not enabled';
        iStep := 8000;
    END_IF
END_IF


CASE iStep OF
    0: (* idle *)
        ;

    (* Get all statuses *)
    10: (* Pumping Station *)
            fbPfeifferTransaction.i_xExecute:= TRUE;
            fbPfeifferTransaction.i_xActionCommand:= FALSE;
            fbPfeifferTransaction.i_iParameterNum:= 10;
            fbPfeifferTransaction.i_iDataLength:= 2;
            fbPfeifferTransaction.i_sSendData:= '=?';
        IF fbPfeifferTransaction.q_xError THEN
            q_sResult := CONCAT('in Step 10 fbPfeifferTransaction failed with message: ', fbPfeifferTransaction.q_sResult);
            iStep := 9000;
        ELSIF fbPfeifferTransaction.q_xDone THEN
            IF fbPfeifferTransaction.q_sResponseData = '000000' OR fbPfeifferTransaction.q_sResponseData = '111111' THEN
                q_stStatus.xPumpingStation_010 := (fbPfeifferTransaction.q_sResponseData = '111111');
                a_ClearTrans();  (* to provide rising edge for execute *)
                iStep := iStep + 10;
            ELSE
                q_sResult := CONCAT('In step 10 invalid data returned from Pfeiffer: ', fbPfeifferTransaction.q_sResponseData);
                iStep := 9000;
            END_IF
        END_IF

    20: (* Gas Mode *)
            fbPfeifferTransaction.i_xExecute:= TRUE;
            fbPfeifferTransaction.i_xActionCommand:= FALSE;
            fbPfeifferTransaction.i_iParameterNum:= 27;
            fbPfeifferTransaction.i_iDataLength:= 2;
            fbPfeifferTransaction.i_sSendData:= '=?';
        IF fbPfeifferTransaction.q_xError THEN
            q_sResult := CONCAT('in Step 20 fbPfeifferTransaction failed with message: ', fbPfeifferTransaction.q_sResult);
            iStep := 9000;
        ELSIF fbPfeifferTransaction.q_xDone THEN
            q_stStatus.iGasMode_027 := STRING_TO_INT( fbPfeifferTransaction.q_sResponseData);
            a_ClearTrans();  (* to provide rising edge for execute *)
            iStep := iStep + 10;
        END_IF

    30: (* Error Code *)
            fbPfeifferTransaction.i_xExecute:= TRUE;
            fbPfeifferTransaction.i_xActionCommand:= FALSE;
            fbPfeifferTransaction.i_iParameterNum:= 303;
            fbPfeifferTransaction.i_iDataLength:= 2;
            fbPfeifferTransaction.i_sSendData:= '=?';
        IF fbPfeifferTransaction.q_xError THEN
            q_sResult := CONCAT('in Step 30 fbPfeifferTransaction failed with message: ', fbPfeifferTransaction.q_sResult);
            iStep := 9000;
        ELSIF fbPfeifferTransaction.q_xDone THEN
            q_stStatus.sErrorCode_303 := fbPfeifferTransaction.q_sResponseData;
            IF LEFT(q_stStatus.sErrorCode_303, 3) = 'Err' THEN
                q_stStatus.iErrorCode_303 := STRING_TO_INT(	RIGHT(q_stStatus.sErrorCode_303, 3) );
                q_stStatus.iWarningCode_303 := 0;
            ELSIF LEFT(q_stStatus.sErrorCode_303, 3) = 'Wrn' THEN
                q_stStatus.iWarningCode_303 := STRING_TO_INT(	RIGHT(q_stStatus.sErrorCode_303, 3) );
                q_stStatus.iErrorCode_303 := 0;
            ELSIF q_stStatus.sErrorCode_303 = '000000' THEN
                q_stStatus.iErrorCode_303 := q_stStatus.iWarningCode_303 := 0;
            END_IF

            a_ClearTrans();  (* to provide rising edge for execute *)
            iStep := iStep + 10;
        END_IF

    40: (* Excess Temperature Pump *)
            fbPfeifferTransaction.i_xExecute:= TRUE;
            fbPfeifferTransaction.i_xActionCommand:= FALSE;
            fbPfeifferTransaction.i_iParameterNum:= 305;
            fbPfeifferTransaction.i_iDataLength:= 2;
            fbPfeifferTransaction.i_sSendData:= '=?';
        IF fbPfeifferTransaction.q_xError THEN
            q_sResult := CONCAT('in Step 40 fbPfeifferTransaction failed with message: ', fbPfeifferTransaction.q_sResult);
            iStep := 9000;
        ELSIF fbPfeifferTransaction.q_xDone THEN
            IF fbPfeifferTransaction.q_sResponseData = '000000' OR fbPfeifferTransaction.q_sResponseData = '111111' THEN
                q_stStatus.xExcessTempPump_305 := (fbPfeifferTransaction.q_sResponseData = '111111');
                a_ClearTrans();  (* to provide rising edge for execute *)
                iStep := iStep + 10;
            ELSE
                q_sResult := CONCAT('In step 40 invalid data returned from Pfeiffer: ', fbPfeifferTransaction.q_sResponseData);
                iStep := 9000;
            END_IF
        END_IF

    50: (* Rotation Speed Attained *)
            fbPfeifferTransaction.i_xExecute:= TRUE;
            fbPfeifferTransaction.i_xActionCommand:= FALSE;
            fbPfeifferTransaction.i_iParameterNum:= 306;
            fbPfeifferTransaction.i_iDataLength:= 2;
            fbPfeifferTransaction.i_sSendData:= '=?';
        IF fbPfeifferTransaction.q_xError THEN
            q_sResult := CONCAT('in Step 50 fbPfeifferTransaction failed with message: ', fbPfeifferTransaction.q_sResult);
            iStep := 9000;
        ELSIF fbPfeifferTransaction.q_xDone THEN
            IF fbPfeifferTransaction.q_sResponseData = '000000' OR fbPfeifferTransaction.q_sResponseData = '111111' THEN
                q_stStatus.xRotationSpeedAttn_306 := (fbPfeifferTransaction.q_sResponseData = '111111');
                a_ClearTrans();  (* to provide rising edge for execute *)
                iStep := iStep + 10;
            ELSE
                q_sResult := CONCAT('In step 50 invalid data returned from Pfeiffer: ', fbPfeifferTransaction.q_sResponseData);
                iStep := 9000;
            END_IF
        END_IF

    60: (* Pump Accelerating *)
            fbPfeifferTransaction.i_xExecute:= TRUE;
            fbPfeifferTransaction.i_xActionCommand:= FALSE;
            fbPfeifferTransaction.i_iParameterNum:= 307;
            fbPfeifferTransaction.i_iDataLength:= 2;
            fbPfeifferTransaction.i_sSendData:= '=?';
        IF fbPfeifferTransaction.q_xError THEN
            q_sResult := CONCAT('in Step 60 fbPfeifferTransaction failed with message: ', fbPfeifferTransaction.q_sResult);
            iStep := 9000;
        ELSIF fbPfeifferTransaction.q_xDone THEN
            IF fbPfeifferTransaction.q_sResponseData = '000000' OR fbPfeifferTransaction.q_sResponseData = '111111' THEN
                q_stStatus.xPumpAccelerating_307 := (fbPfeifferTransaction.q_sResponseData = '111111');
                a_ClearTrans();  (* to provide rising edge for execute *)
                iStep := iStep + 10;
            ELSE
                q_sResult := CONCAT('In step 60 invalid data returned from Pfeiffer: ', fbPfeifferTransaction.q_sResponseData);
                iStep := 9000;
            END_IF
        END_IF

    70: (* Acitve Rotation Speed *)
            fbPfeifferTransaction.i_xExecute:= TRUE;
            fbPfeifferTransaction.i_xActionCommand:= FALSE;
            fbPfeifferTransaction.i_iParameterNum:= 309;
            fbPfeifferTransaction.i_iDataLength:= 2;
            fbPfeifferTransaction.i_sSendData:= '=?';
        IF fbPfeifferTransaction.q_xError THEN
            q_sResult := CONCAT('in Step 70 fbPfeifferTransaction failed with message: ', fbPfeifferTransaction.q_sResult);
            iStep := 9000;
        ELSIF fbPfeifferTransaction.q_xDone THEN
            q_stStatus.diActiveRotationSpeed_309 := STRING_TO_DINT( fbPfeifferTransaction.q_sResponseData);
            a_ClearTrans();  (* to provide rising edge for execute *)
            iStep := iStep + 1;
        END_IF

    71: (* Electronics Temp *)
            fbPfeifferTransaction.i_xExecute:= TRUE;
            fbPfeifferTransaction.i_xActionCommand:= FALSE;
            fbPfeifferTransaction.i_iParameterNum:= 326;
            fbPfeifferTransaction.i_iDataLength:= 2;
            fbPfeifferTransaction.i_sSendData:= '=?';
        IF fbPfeifferTransaction.q_xError THEN
            q_sResult := CONCAT('in Step 71 fbPfeifferTransaction failed with message: ', fbPfeifferTransaction.q_sResult);
            iStep := 9000;
        ELSIF fbPfeifferTransaction.q_xDone THEN
            q_stStatus.diTempElec_326 := STRING_TO_DINT( fbPfeifferTransaction.q_sResponseData);
            a_ClearTrans();  (* to provide rising edge for execute *)
            iStep := iStep + 1;
        END_IF

    72: (* Bottom of Pump Temp *)
            fbPfeifferTransaction.i_xExecute:= TRUE;
            fbPfeifferTransaction.i_xActionCommand:= FALSE;
            fbPfeifferTransaction.i_iParameterNum:= 330;
            fbPfeifferTransaction.i_iDataLength:= 2;
            fbPfeifferTransaction.i_sSendData:= '=?';
        IF fbPfeifferTransaction.q_xError THEN
            q_sResult := CONCAT('in Step 72 fbPfeifferTransaction failed with message: ', fbPfeifferTransaction.q_sResult);
            iStep := 9000;
        ELSIF fbPfeifferTransaction.q_xDone THEN
            q_stStatus.diTempPmpBot_330 := STRING_TO_DINT( fbPfeifferTransaction.q_sResponseData);
            a_ClearTrans();  (* to provide rising edge for execute *)
            iStep := iStep + 1;
        END_IF

    73: (* Temp bearing *)
            fbPfeifferTransaction.i_xExecute:= TRUE;
            fbPfeifferTransaction.i_xActionCommand:= FALSE;
            fbPfeifferTransaction.i_iParameterNum:= 342;
            fbPfeifferTransaction.i_iDataLength:= 2;
            fbPfeifferTransaction.i_sSendData:= '=?';
        IF fbPfeifferTransaction.q_xError THEN
            q_sResult := CONCAT('in Step 73 fbPfeifferTransaction failed with message: ', fbPfeifferTransaction.q_sResult);
            iStep := 9000;
        ELSIF fbPfeifferTransaction.q_xDone THEN
            q_stStatus.diTempBearng_342 := STRING_TO_DINT( fbPfeifferTransaction.q_sResponseData);
            a_ClearTrans();  (* to provide rising edge for execute *)
            iStep := iStep + 1;
        END_IF


    74: (* Temp motor *)
            fbPfeifferTransaction.i_xExecute:= TRUE;
            fbPfeifferTransaction.i_xActionCommand:= FALSE;
            fbPfeifferTransaction.i_iParameterNum:= 346;
            fbPfeifferTransaction.i_iDataLength:= 2;
            fbPfeifferTransaction.i_sSendData:= '=?';
        IF fbPfeifferTransaction.q_xError THEN
            q_sResult := CONCAT('in Step 74 fbPfeifferTransaction failed with message: ', fbPfeifferTransaction.q_sResult);
            iStep := 9000;
        ELSIF fbPfeifferTransaction.q_xDone THEN
            q_stStatus.diTempMotor_346 := STRING_TO_DINT( fbPfeifferTransaction.q_sResponseData);
            a_ClearTrans();  (* to provide rising edge for execute *)
            iStep := 80;
        END_IF

    80: (* Drive Current *)
            fbPfeifferTransaction.i_xExecute:= TRUE;
            fbPfeifferTransaction.i_xActionCommand:= FALSE;
            fbPfeifferTransaction.i_iParameterNum:= 310;
            fbPfeifferTransaction.i_iDataLength:= 2;
            fbPfeifferTransaction.i_sSendData:= '=?';
        IF fbPfeifferTransaction.q_xError THEN
            q_sResult := CONCAT('in Step 80 fbPfeifferTransaction failed with message: ', fbPfeifferTransaction.q_sResult);
            iStep := 9000;
        ELSIF fbPfeifferTransaction.q_xDone THEN
            q_stStatus.lrDriveCurrent_310 := STRING_TO_LREAL( fbPfeifferTransaction.q_sResponseData)/100.0;
            a_ClearTrans();  (* to provide rising edge for execute *)
            iStep := iStep + 10;
        END_IF

    90: (* Drive Power *)
            fbPfeifferTransaction.i_xExecute:= TRUE;
            fbPfeifferTransaction.i_xActionCommand:= FALSE;
            fbPfeifferTransaction.i_iParameterNum:= 316;
            fbPfeifferTransaction.i_iDataLength:= 2;
            fbPfeifferTransaction.i_sSendData:= '=?';
        IF fbPfeifferTransaction.q_xError THEN
            q_sResult := CONCAT('in Step 90 fbPfeifferTransaction failed with message: ', fbPfeifferTransaction.q_sResult);
            iStep := 9000;
        ELSIF fbPfeifferTransaction.q_xDone THEN
            q_stStatus.diDrivePower_316 := STRING_TO_DINT( fbPfeifferTransaction.q_sResponseData);
            a_ClearTrans();  (* to provide rising edge for execute *)
            iStep := 91;
        END_IF

    91: (* Check Power Consumption Limit *)
            fbPfeifferTransaction.i_xExecute:= TRUE;
            fbPfeifferTransaction.i_xActionCommand:= FALSE;
            fbPfeifferTransaction.i_iParameterNum:= 708;
            fbPfeifferTransaction.i_iDataLength:= 2;
            fbPfeifferTransaction.i_sSendData:= '=?';
        IF fbPfeifferTransaction.q_xError THEN
            q_sResult := CONCAT('in Step 91 fbPfeifferTransaction failed with message: ', fbPfeifferTransaction.q_sResult);
            iStep := 9000;
        ELSIF fbPfeifferTransaction.q_xDone THEN
            q_stStatus.uiPowerPct_708 := STRING_TO_UINT( fbPfeifferTransaction.q_sResponseData);
            a_ClearTrans();  (* to provide rising edge for execute *)
            iStep := 8000;// this step not tested 110; // was 5000, but we don't want to control via serial but via PLC IO, just write the pump speed
        END_IF

    100:
        (*IF (i_stControl.iSetRotationSpeed_707 <> diOldSetRotationSpeed_707) AND ( i_stControl.iSetRotationSpeed_707 <> 0)  THEN
            diOldSetRotationSpeed_707 := i_stControl.iSetRotationSpeed_707;
            iStep := 110;
        ELSE
            q_sResult := 'Success';
            iStep := 8000;// maybe should be 5000
        END_IF*)

    110: (* Set  SpdSetMode: Rotation speed setting mode*)
        IF i_stControl.xSetSpdMode_026 THEN
            sSendData := '001';
        ELSE
            sSendData := '000';
        END_IF
            //i_stControl.iSetSpdMode_026:=1;
            //fbFormatString( sFormat:= '%.3u', arg1:= F_INT(i_stControl.iSetSpdMode_026), sOut => sSendData);
            fbPfeifferTransaction.i_xExecute:= TRUE;
            fbPfeifferTransaction.i_xActionCommand:= TRUE;
            fbPfeifferTransaction.i_iParameterNum:= 26;
            fbPfeifferTransaction.i_iDataLength:= 3;
            fbPfeifferTransaction.i_sSendData:= sSendData;
        IF fbPfeifferTransaction.q_xError THEN
            q_sResult := CONCAT('in Step 110 fbPfeifferTransaction failed with message: ', fbPfeifferTransaction.q_sResult);
            iStep := 9000;
        ELSIF fbPfeifferTransaction.q_xDone THEN
            IF fbPfeifferTransaction.q_sResponseData = sSendData THEN
                q_stStatus.iSetSpdMode_026 := STRING_TO_INT(fbPfeifferTransaction.q_sResponseData);
                a_ClearTrans();  (* to provide rising edge for execute *)
                iStep := 120;
            ELSE
                q_sResult := CONCAT('In step 110 invalid data returned from Pfeiffer: ', fbPfeifferTransaction.q_sResponseData);
                iStep := 9000;
            END_IF
        END_IF

    120:(* Update Pump Speed *) (* SpdSVal % Set value in rot. speed setting mode *)
            i_stControl.iSetRotationSpeed_707 := i_stControl.iSetRotationSpeed_707 *100; //Datatype 2
            fbFormatString( sFormat:= '%.6u', arg1:= F_INT(i_stControl.iSetRotationSpeed_707), sOut => sSendData);
            fbPfeifferTransaction.i_xExecute:= TRUE;
            fbPfeifferTransaction.i_xActionCommand:= TRUE;
            fbPfeifferTransaction.i_iParameterNum:= 707;
            fbPfeifferTransaction.i_iDataLength:= 6;
            fbPfeifferTransaction.i_sSendData:= sSendData;
        IF fbPfeifferTransaction.q_xError THEN
            q_sResult := CONCAT('in Step 120 fbPfeifferTransaction failed with message: ', fbPfeifferTransaction.q_sResult);
            iStep := 9000;
        ELSIF fbPfeifferTransaction.q_xDone THEN
            IF fbPfeifferTransaction.q_sResponseData = sSendData THEN
            q_stStatus.iSetRotationSpeed_707 := STRING_TO_INT( fbPfeifferTransaction.q_sResponseData);
                a_ClearTrans();  (* to provide rising edge for execute *)
                iStep := 8000;
            ELSE
                q_sResult := CONCAT('In step 120 invalid data returned from Pfeiffer: ', fbPfeifferTransaction.q_sResponseData);
                iStep := 9000;
            END_IF
        END_IF


    130: (* Set  SpdSetMode: Rotation speed setting mode Off*)
        (*	i_stControl.iSetSpdMode_026:=0;
            fbFormatString( sFormat:= '%.3u', arg1:= F_INT(i_stControl.iSetSpdMode_026), sOut => sSendData);
            fbPfeifferTransaction.i_xExecute:= TRUE;
            fbPfeifferTransaction.i_xActionCommand:= TRUE;
            fbPfeifferTransaction.i_iParameterNum:= 26;
            fbPfeifferTransaction.i_iDataLength:= 3;
            fbPfeifferTransaction.i_sSendData:= sSendData;
        IF fbPfeifferTransaction.q_xError THEN
            q_sResult := CONCAT('in Step 110 fbPfeifferTransaction failed with message: ', fbPfeifferTransaction.q_sResult);
            iStep := 9000;
        ELSIF fbPfeifferTransaction.q_xDone THEN
            IF fbPfeifferTransaction.q_sResponseData = sSendData THEN
                q_stStatus.iSetSpdMode_026 := STRING_TO_INT(fbPfeifferTransaction.q_sResponseData);
                a_ClearTrans();  (* to provide rising edge for execute *)
                iStep := 100;
            ELSE
                q_sResult := CONCAT('In step 110 invalid data returned from Pfeiffer: ', fbPfeifferTransaction.q_sResponseData);
                iStep := 9000;
            END_IF
        END_IF*)

    5000:(* Check Status vs. requested parameters, set iff necessary *)
        IF i_stControl.xErrorAck_009 THEN
            iStep := 5030;
        ELSIF i_stControl.xPumpingStation_010 <> q_stStatus.xPumpingStation_010 THEN
            //iStep := 5010; Done through the PLC DIO
        ELSIF  i_stControl.iGasMode_027 <> q_stStatus.iGasMode_027 THEN
            iStep := 5020;
        ELSIF i_stControl.xMotorPump_023 <> q_stStatus.xMotorPump_023 THEN
            //iStep := 5011;  Done through the PLC DIO
        ELSIF i_stControl.uiPowerPct_708 <> q_stStatus.uiPowerPct_708 THEN
            iStep := 5012;
        ELSE
            q_sResult := 'Success';
            iStep := 8000;
        END_IF

    5010: (* Update Pumping Station *)
        IF i_stControl.xPumpingStation_010 THEN
            sSendData := '111111';
        ELSE
            sSendData := '000000';
        END_IF
            fbPfeifferTransaction.i_xExecute:= TRUE;
            fbPfeifferTransaction.i_xActionCommand:= TRUE;
            fbPfeifferTransaction.i_iParameterNum:= 10;
            fbPfeifferTransaction.i_iDataLength:= 6;
            fbPfeifferTransaction.i_sSendData:= sSendData;
        IF fbPfeifferTransaction.q_xError THEN
            q_sResult := CONCAT('in Step 5010 fbPfeifferTransaction failed with message: ', fbPfeifferTransaction.q_sResult);
            iStep := 9000;
        ELSIF fbPfeifferTransaction.q_xDone THEN
            IF fbPfeifferTransaction.q_sResponseData = sSendData THEN
                q_stStatus.xPumpingStation_010 := (fbPfeifferTransaction.q_sResponseData = '111111');
                a_ClearTrans();  (* to provide rising edge for execute *)
                iStep := 5000;
            ELSE
                q_sResult := CONCAT('In step 5010 invalid data returned from Pfeiffer: ', fbPfeifferTransaction.q_sResponseData);
                iStep := 9000;
            END_IF
        END_IF

    5011: (* Update Pump Motor *)
        IF i_stControl.xMotorPump_023 THEN
            sSendData := '111111';
        ELSE
            sSendData := '000000';
        END_IF
            fbPfeifferTransaction.i_xExecute:= TRUE;
            fbPfeifferTransaction.i_xActionCommand:= TRUE;
            fbPfeifferTransaction.i_iParameterNum:= 23;
            fbPfeifferTransaction.i_iDataLength:= 6;
            fbPfeifferTransaction.i_sSendData:= sSendData;
        IF fbPfeifferTransaction.q_xError THEN
            q_sResult := CONCAT('in Step 5011 fbPfeifferTransaction failed with message: ', fbPfeifferTransaction.q_sResult);
            iStep := 9000;
        ELSIF fbPfeifferTransaction.q_xDone THEN
            IF fbPfeifferTransaction.q_sResponseData = sSendData THEN
                q_stStatus.xMotorPump_023 := (fbPfeifferTransaction.q_sResponseData = '111111');
                a_ClearTrans();  (* to provide rising edge for execute *)
                iStep := 5000;
            ELSE
                q_sResult := CONCAT('In step 5011 invalid data returned from Pfeiffer: ', fbPfeifferTransaction.q_sResponseData);
                iStep := 9000;
            END_IF
        END_IF

    5012: (* Update Power Consumption Percent *)
        fbFormatString( sFormat:= '%.6u', arg1:= F_UINT(i_stControl.uiPowerPct_708), sOut => sSendData);
            fbPfeifferTransaction.i_xExecute:= TRUE;
            fbPfeifferTransaction.i_xActionCommand:= TRUE;
            fbPfeifferTransaction.i_iParameterNum:= 708;
            fbPfeifferTransaction.i_iDataLength:= 3;
            fbPfeifferTransaction.i_sSendData:= sSendData;
        IF fbPfeifferTransaction.q_xError THEN
            q_sResult := CONCAT('in Step 5012 fbPfeifferTransaction failed with message: ', fbPfeifferTransaction.q_sResult);
            iStep := 9000;
        ELSIF fbPfeifferTransaction.q_xDone THEN
            IF fbPfeifferTransaction.q_sResponseData = sSendData THEN
                q_stStatus.uiPowerPct_708 := STRING_TO_UINT(fbPfeifferTransaction.q_sResponseData);
                a_ClearTrans();  (* to provide rising edge for execute *)
                iStep := 5000;
            ELSE
                q_sResult := CONCAT('In step 5012 invalid data returned from Pfeiffer: ', fbPfeifferTransaction.q_sResponseData);
                iStep := 9000;
            END_IF
        END_IF

    5020: (* Update Gas Mode *)
        fbFormatString( sFormat:= '%.3u', arg1:= F_INT(i_stControl.iGasMode_027), sOut => sSendData);
            fbPfeifferTransaction.i_xExecute:= TRUE;
            fbPfeifferTransaction.i_xActionCommand:= TRUE;
            fbPfeifferTransaction.i_iParameterNum:= 27;
            fbPfeifferTransaction.i_iDataLength:= 3;
            fbPfeifferTransaction.i_sSendData:= sSendData;
        IF fbPfeifferTransaction.q_xError THEN
            q_sResult := CONCAT('in Step 5020 fbPfeifferTransaction failed with message: ', fbPfeifferTransaction.q_sResult);
            iStep := 9000;
        ELSIF fbPfeifferTransaction.q_xDone THEN
            IF fbPfeifferTransaction.q_sResponseData = sSendData THEN
                q_stStatus.iGasMode_027 := STRING_TO_INT(fbPfeifferTransaction.q_sResponseData);
                a_ClearTrans();  (* to provide rising edge for execute *)
                iStep := 5000;
            ELSE
                q_sResult := CONCAT('In step 5020 invalid data returned from Pfeiffer: ', fbPfeifferTransaction.q_sResponseData);
                iStep := 9000;
            END_IF
        END_IF

    5030: (* Update Error Acknowledgement *)
        IF i_stControl.xErrorAck_009 THEN
            q_stStatus.xErrorAcknowledged := TRUE;
            sSendData := '111111';
        ELSE
            sSendData := '000000';
        END_IF
            fbPfeifferTransaction.i_xExecute:= TRUE;
            fbPfeifferTransaction.i_xActionCommand:= TRUE;
            fbPfeifferTransaction.i_iParameterNum:= 9;
            fbPfeifferTransaction.i_iDataLength:= 6;
            fbPfeifferTransaction.i_sSendData:= sSendData;
        IF fbPfeifferTransaction.q_xError THEN
            q_sResult := CONCAT('in Step 5030 fbPfeifferTransaction failed with message: ', fbPfeifferTransaction.q_sResult);
            iStep := 9000;
        ELSIF fbPfeifferTransaction.q_xDone THEN (* Error Acknowledged *)
                a_ClearTrans();  (* to provide rising edge for execute *)
                iStep := 5000;
        END_IF


    8000: (* done *)
        q_xDone := TRUE;
        a_ClearTrans();  (* to provide rising edge for execute *)
        IF  i_xExecute = FALSE THEN
            q_xDone:= FALSE;
            iStep := 0;
        END_IF

    9000:
        _A_ClearStatus();
        a_ClearTrans();  (* to provide rising edge for execute *)
        q_xError := TRUE;

END_CASE

//call transaction
fbPfeifferTransaction(
    i_iAddress:= i_stControl.iSerialAddress,
    i_tTimeOut:= i_tTimeOut,
    iq_stSerialRXBuffer:= iq_stSerialRXBuffer,
    iq_stSerialTXBuffer:= iq_stSerialTXBuffer );

q_stStatus.xTimeout := fbPfeifferTransaction.q_xTimeout;
q_sLastSentString := fbPfeifferTransaction.q_sLastSentString;
q_sLastReceivedString := fbPfeifferTransaction.q_sLastReceivedString;

ACTION _A_ClearStatus:
q_stStatus.xPumpingStation_010 := FALSE;
q_stStatus.iGasMode_027 := 0;
q_stStatus.sErrorCode_303 := '';
q_stStatus.xExcessTempPump_305 := FALSE;
q_stStatus.xRotationSpeedAttn_306 := FALSE;
q_stStatus.xPumpAccelerating_307 := FALSE;
q_stStatus.diActiveRotationSpeed_309 := 0;
q_stStatus.lrDriveCurrent_310 := 0;
q_stStatus.diDrivePower_316 := 0;
END_ACTION

ACTION a_ClearTrans:
fbPfeifferTransaction.i_xExecute := FALSE;
fbPfeifferTransaction.i_xActionCommand:= FALSE;
fbPfeifferTransaction.i_iParameterNum:= 0;
fbPfeifferTransaction.i_iDataLength:= 0;
fbPfeifferTransaction.i_sSendData:= '';
END_ACTION

END_FUNCTION_BLOCK

// ---- POUs/Serial drivers/Pumps/Pfeiffer/FB_PfeifferTransaction.TcPOU
FUNCTION_BLOCK FB_PfeifferTransaction
VAR_INPUT
    /// rising edge execute
    i_xExecute: BOOL;
    /// RS-485 Address of Pump
    i_iAddress: INT;
    /// False is data request, True is control command
    i_xActionCommand: BOOL;
    /// Parameter Number 1-999
    i_iParameterNum: INT;
    /// Send Data Length
    i_iDataLength: INT;
    /// Send Data
    i_sSendData: STRING;
    /// Maximum wait time for reply
    i_tTimeOut: TIME := TIME#1s0ms;
END_VAR
VAR_OUTPUT
    q_xDone: BOOL;
    q_sResponseData: STRING;
    q_xError: BOOL;
    q_xTimeout: BOOL;
    q_sResult: STRING;
    /// Last String Sent to Serial Device - for debugging
    q_sLastSentString: STRING;
    /// Last String Received from Serial Device - for debugging
    q_sLastReceivedString: STRING;
END_VAR
VAR_IN_OUT
    iq_stSerialRXBuffer: ComBuffer;
    iq_stSerialTXBuffer: ComBuffer;
END_VAR
VAR
    rtExecute: R_TRIG;
    iStep: INT;
    fbClearComBuffer: ClearComBuffer;
    sSendString: STRING;
    fbFormatString: FB_FormatString;
    iChecksum: INT;
    fbSendString: SendString;
    fbReceiveString: ReceiveString;
    sReceivedString: STRING;
    tonTimeout: TON;
    sRXStringForChecksum: STRING;
    sReceiveStringWOChecksum: STRING;
    sRXCheckSum: STRING;
    sRXAddress: STRING;
    sRXParmNum: STRING;
END_VAR

(* This function block performs serial transactions with a Pfeiffer RC400 Pump controller *)

(* rising edge trigger *)
rtExecute(CLK:= i_xExecute);
IF rtExecute.Q THEN
    q_xDone	:= FALSE;
    q_sResponseData := '';
    q_xError := FALSE;
    //q_xTimeout := FALSE;
    q_sResult:= '';
    q_sLastSentString := '';
    q_sLastReceivedString:= '';
    iStep := 10;
END_IF

CASE iStep OF
    0:
        ; (* idle *)

    10: (* clear com buffers *)
        fbClearComBuffer(Buffer:= iq_stSerialRXBuffer);
        fbClearComBuffer(Buffer:= iq_stSerialTXBuffer);

        (* build the send string *)
        fbFormatString( sFormat:= '%0.3d', arg1:= F_INT(i_iAddress), sOut=> sSendString); (* address *)
        IF i_xActionCommand THEN (* action *)
            sSendString := CONCAT(sSendString, '10');
        ELSE
            sSendString := CONCAT(sSendString, '00');
        END_IF
        fbFormatString( sFormat:= '%0.3u', arg1:= F_INT(i_iParameterNum)); (* parameter number *)
        sSendString := CONCAT(sSendString, fbFormatString.sOut);
        fbFormatString( sFormat:= '%0.2u', arg1:= F_INT(i_iDataLength)); (* data length *)
        sSendString := CONCAT(sSendString, fbFormatString.sOut);
        sSendString := CONCAT(sSendString, i_sSendData); (* data *)
        iChecksum := F_CalcPfeifferChecksum(sSendString); (* checksum *)
        fbFormatString( sFormat:= '%0.3u$R', arg1:= F_INT(iChecksum));
        sSendString := CONCAT(sSendString, fbFormatString.sOut);
        (* send it *)
        fbSendString( SendString:= sSendString, TXbuffer:= iq_stSerialTXBuffer );
        q_sLastSentString := sSendString;
        iStep := iStep + 10;

    20: (* Finish sending the String *)
        IF fbSendString.Busy THEN
            fbSendString( SendString:= sSendString, TXbuffer:= iq_stSerialTXBuffer );
        ELSIF fbSendString.Error <> 0 THEN
            q_sResult := CONCAT('In step 20 fbSendString resulted in error: ', INT_TO_STRING(fbSendString.Error));
            iStep := 9000;
        ELSIF NOT fbSendString.Busy THEN
            iStep := iStep + 10;
        END_IF
        (* Reset receive *)
        fbReceiveString(
            Reset:= TRUE,
            ReceivedString:= sReceivedString,
            RXbuffer:= iq_stSerialRXBuffer );
        tonTimeout(IN:= FALSE);

    30: (* Get reply *)
        fbReceiveString(
            Prefix:= ,
            Suffix:= '$R',
            Timeout:= i_tTimeOut,
            Reset:= FALSE,
            ReceivedString:= sReceivedString,
            RXbuffer:= iq_stSerialRXBuffer );
        tonTimeout(IN:= TRUE, PT:= i_tTimeOut);
        IF fbReceiveString.Error <> 0 AND fbReceiveString.Error <> 16#1008 THEN //16#1008 is timeout error
            q_sResult := CONCAT('In step 30 fbReceiveString resulted in error: ', INT_TO_STRING(fbReceiveString.Error));
            iStep := 9000;
        ELSIF fbReceiveString.RxTimeout OR tonTimeout.Q THEN
            q_sResult := 'Pfeiffer pump failed to reply within timeout period';
            q_xTimeout := TRUE;
            iStep := 9000;
        ELSIF fbReceiveString.StringReceived THEN
            q_xTimeout := FALSE; //no timeout
            q_sLastReceivedString := sReceivedString;
            (* check checksum *)
            sReceiveStringWOChecksum := LEFT(sReceivedString, LEN(sReceivedString)-4);
            iChecksum := F_CalcPfeifferChecksum(sReceiveStringWOChecksum);
            sRXCheckSum := MID(sReceivedString,3,LEN(sReceivedString)-3);
            sRXAddress := LEFT(sReceivedString,3);
            sRXParmNum := MID(sReceivedString,3,6);
            IF iChecksum <> STRING_TO_INT(sRXCheckSum) THEN
                q_sResult := 'Invalid checksum on received string.';
                iStep := 9000;
            ELSIF i_iAddress <> STRING_TO_INT(sRXAddress) THEN
                q_sResult := 'Invalid unit address on received string.';
                iStep := 9000;
            ELSIF i_iParameterNum <> STRING_TO_INT(sRXParmNum) THEN
                q_sResult := 'Invalid parameter number on received string.';
                iStep := 9000;
            ELSE
                q_sResponseData := MID(sReceivedString,LEN(sReceivedString)-14 ,11);
                q_sResult := 'Success.';
                q_xDone:= TRUE;
                iStep := 100;
            END_IF
        END_IF

    100: (* done *)
        IF  i_xExecute = FALSE THEN
            q_xDone:= FALSE;
            iStep := 0;
        END_IF

    9000:
        q_xError := TRUE;




END_CASE

END_FUNCTION_BLOCK

// ---- POUs/Serial drivers/Pumps/Pfeiffer/F_CalcPfeifferCheckSum.TcPOU
FUNCTION F_CalcPfeifferCheckSum : BYTE
VAR_INPUT
    sData: STRING;
END_VAR
VAR
    bSum: BYTE;
    i: INT;
END_VAR

bSum := 0;

FOR i := 1 TO LEN(sData) DO
    bSum := bSum + F_ToASC(MID(sData,1,i));
END_FOR

F_CalcPfeifferChecksum := bSum;

END_FUNCTION

// ---- POUs/Serial drivers/Pumps/Pfeiffer/FB_PFEIFFER_COM.TcPOU
FUNCTION_BLOCK FB_PFEIFFER_COM
VAR_IN_OUT
    astPfeifferControl: ARRAY[1..gcMaxPfeifferPumps] OF ST_PfeifferControl;
    astPfeifferStatus: ARRAY[1..gcMaxPfeifferPumps] OF ST_PfeifferStatus;
    SerialRXBuffer: ComBuffer;
    SerialTXBuffer: ComBuffer;
END_VAR
VAR
    afbPfeifferSerialDriver: ARRAY[1..gcMaxPfeifferPumps] OF FB_PfeifferSerialDriver;
    iPump: INT := 1;
    tTimeOut: TIME := TIME#1s0ms;
END_VAR

(* This program is called from Serial PTM IO *)

(* scan the pumps one at a time *)
afbPfeifferSerialDriver[iPump](
    i_xExecute:= TRUE,
    i_tTimeOut:= tTimeOut,
    i_stControl:=astPfeifferControl[iPump] ,
    iq_stSerialRXBuffer:= SerialRXBuffer,
    iq_stSerialTXBuffer:=  SerialTXBuffer,
    q_stStatus=> astPfeifferStatus[iPump] );

IF afbPfeifferSerialDriver[iPump].q_xDone
OR afbPfeifferSerialDriver[iPump].q_xError
THEN
        (* reset for next time *)
        afbPfeifferSerialDriver[iPump]( i_xExecute:= FALSE, iq_stSerialRXBuffer:= SerialRXBuffer, iq_stSerialTXBuffer:=  SerialTXBuffer);
        (* select next pump *)
        iPump := iPump + 1;
        IF iPump > gcMaxPfeifferPumps THEN
            iPump:= 1;
        END_IF
END_IF

END_FUNCTION_BLOCK

// ---- POUs/Serial drivers/Pumps/Pfeiffer/FB_PFEIFFER_TO_PTM.TcPOU
FUNCTION_BLOCK FB_PFEIFFER_TO_PTM
VAR_IN_OUT
    {attribute 'pytmc' :=' pv:'}
    iq_stPTM: ST_PfeifferPTM;
    iq_stPfeiffer_ctrl: ST_PfeifferControl;
    iq_stPfeiffer_stat: ST_PfeifferStatus;
END_VAR

(* This function block is used to map the IO points from the pfeiffer structures
to the generic turbo structures *)

(* Controls *)
iq_stPfeiffer_ctrl.xPumpingStation_010 := iq_stPTM.q_RunDO;
iq_stPfeiffer_ctrl.xMotorPump_023 := 1; //Setting always true because parameter 10 alone can enable/disable the pump
iq_stPfeiffer_ctrl.uiPowerPct_708 := iq_stPTM.q_uiPowerPct;
iq_stPfeiffer_ctrl.xErrorAck_009 := iq_stPTM.xResetSW;

(* Readbacks *)
iq_stPTM.i_xAccel := iq_stPfeiffer_stat.xPumpAccelerating_307;
iq_stPTM.i_xAtSpd := iq_stPfeiffer_stat.xRotationSpeedAttn_306;
iq_stPTM.i_diCurSpd := iq_stPfeiffer_stat.diActiveRotationSpeed_309;
iq_stPTM.i_diPwr := iq_stPfeiffer_stat.diDrivePower_316;
iq_stPTM.i_diElecTemp := iq_stPfeiffer_stat.diTempElec_326;
iq_stPTM.i_diBtmTemp := iq_stPfeiffer_stat.diTempPmpBot_330;
iq_stPTM.i_diBrngTemp := iq_stPfeiffer_stat.diTempBearng_342;
iq_stPTM.i_diMtrTemp := iq_stPfeiffer_stat.diTempMotor_346;
iq_stPTM.i_uiPowerPctRbk := iq_stPfeiffer_stat.uiPowerPct_708;

iq_stPTM.xCommTimeout	:=	iq_stPfeiffer_stat.xTimeout;
iq_stPTM.i_iErrorCode := iq_stPfeiffer_stat.iErrorCode_303;
iq_stPTM.i_iWarningCode := iq_stPfeiffer_stat.iWarningCode_303;

(* Check that error acknowledgment is processed*)
IF iq_stPfeiffer_stat.xErrorAcknowledged THEN
    iq_stPfeiffer_stat.xErrorAcknowledged := FALSE;
    iq_stPfeiffer_ctrl.xErrorAck_009 := FALSE;
    iq_stPTM.xResetSW := FALSE;
END_IF

IF iq_stPfeiffer_stat.sErrorCode_303 = '' THEN
    ;
ELSIF iq_stPfeiffer_stat.sErrorCode_303 <> '000000' THEN
iq_stPTM.i_xFault := TRUE;
ELSE
iq_stPTM.i_xFault := FALSE;
END_IF

END_FUNCTION_BLOCK

// ---- UnitTests/Gauges/FB_GCC_Test.TcPOU
FUNCTION_BLOCK FB_GCC_Test EXTENDS TcUnit.FB_TestSuite
VAR_INPUT
END_VAR
VAR_OUTPUT
END_VAR
VAR
    PG : ST_VG;
    fb_MKS422: FB_MKS422;
    //fb_MKS500: FB_MKS500;
    i_iPRESS_R AT %Q* :INT;
    cycle:INT :=0;
END_VAR

M_INIT();
M_Interlock();
M_CheckRange();
//M_SelfProtection();
cycle:=cycle+1;

METHOD M_CheckRange
VAR
    Expected:REAL;
    Actual:REAL;
    eStateExpected: E_PressureState;
    eStateActual: E_PressureState;
END_VAR
TEST('Check_Range');
Case This^.cycle of
    12:
    This^.i_iPRESS_R :=  V_TO_INT(0.61);
    This^.PG.rPRESS := 1E-4;
    This^.PG.xPRESS_OK := True;
    fb_MKS422.M_HVE(TRUE);

    15:
    TEST('MKS422_Range_937B');
    Expected :=1E-11 ;
    eStateExpected := Valid;
    Actual := This^.fb_MKS422.IG.rPRESS;
    eStateActual := This^.fb_MKS422.IG.eState;
    AssertTrue(This^.fb_MKS422.IG.xPRESS_OK, 'MKS422B xPRESS_OK is set to False');
    AssertEquals(eStateExpected,eStateActual,'MKS422B eState Fail');
    AssertEquals_REAL(Expected, Actual,1E-12, 'MKS422B rPress Fail');
    TEST_FINISHED_NAMED('MKS422_Range_937B');

    16:
    This^.i_iPRESS_R := V_TO_INT(2.4);
    This^.fb_MKS422.b937A:=TRUE;

    20:
    TEST('MKS422_Range_937A');
    Expected :=1E-8 ;
    Actual := This^.fb_MKS422.IG.rPRESS;
    eStateExpected := Valid;
    eStateActual := This^.fb_MKS422.IG.eState;
    AssertTrue(This^.fb_MKS422.IG.xPRESS_OK, 'MKS422A xPRESS_OK is set to False');
    AssertEquals(eStateExpected,eStateActual,'MKS422A eState Fail');
    AssertEquals_REAL(Expected, Actual,1E-9, 'MKS422A rPress Fail');
    TEST_FINISHED_NAMED('MKS422_Range_937A');


    21:
    This^.i_iPRESS_R :=  V_TO_INT(0.1);


    24:
    TEST('MKS422_Range_Off');
    Expected :=0 ;
    eStateExpected := GaugeDisconnected;
    Actual := This^.fb_MKS422.IG.rPRESS;
    eStateActual := This^.fb_MKS422.IG.eState;
    AssertFalse(This^.fb_MKS422.IG.xPRESS_OK, 'MKS422A xPRESS_OK is set to True');
    AssertEquals(eStateExpected,eStateActual,'MKS422A eState Fail');
    AssertEquals_REAL(Expected, Actual,1, 'MKS422A rPress Fail');
    TEST_FINISHED_NAMED('MKS422_Range_Off');


    25:
    This^.i_iPRESS_R :=  V_TO_INT(10);


    29:
    TEST('MKS422_Range_Invalid');
    Expected :=0 ;
    eStateExpected := PressInvalid;
    Actual := This^.fb_MKS422.IG.rPRESS;
    eStateActual := This^.fb_MKS422.IG.eState;
    AssertFalse(This^.fb_MKS422.IG.xPRESS_OK, 'MKS422A xPRESS_OK is set to True');
    AssertEquals(eStateExpected,eStateActual,'MKS422A eState Fail');
    AssertEquals_REAL(Expected, Actual,1, 'MKS422A rPress Fail');
    TEST_FINISHED_NAMED('MKS422_Range_Invalid');
    TEST_FINISHED_NAMED('Check_Range');

END_CASE

This^.fb_MKS422(PG:=This^.PG, IG=>);
END_METHOD

METHOD M_INIT
VAR
END_VAR
TEST('MKS422_Startup');
This^.PG.rPRESS := 1E-4;
This^.PG.xPRESS_OK := TRUE;
This^.fb_MKS422(PG:=This^.PG, IG=>);
IF( cycle = 3) THEN
    AssertFalse(This^.fb_MKS422.IG.xHV_SW, 'MKS422 xHV_SW set to True');
    AssertTrue(This^.fb_MKS422.IG.q_xHV_DIS, 'MKS422 q_xHV_DIS set to False');
    TEST_FINISHED_NAMED('MKS422_Startup');
End_IF;
END_METHOD

METHOD M_Interlock
VAR_INPUT
END_VAR
TEST('MKS422_Interlock_Active');
TEST('MKS422_Interlock_OK');
TEST('MKS422_Interlock_Lost');

Case cycle of
    1:
    This^.PG.rPRESS := 1E-1;
    This^.PG.xPRESS_OK := TRUE;
    fb_MKS422.M_HVE(TRUE);

    3:
    AssertFalse(This^.fb_MKS422.IG.xHV_SW, 'MKS422 xHV_SW set to True');
    AssertTrue(This^.fb_MKS422.IG.q_xHV_DIS, 'MKS422 q_xHV_DIS set to False');
    TEST_FINISHED_NAMED('MKS422_Interlock_Active');

    4:
    This^.PG.rPRESS := 1E-4;
    This^.PG.xPRESS_OK := True;
    fb_MKS422.M_HVE(TRUE);

    7:
    AssertTrue(This^.fb_MKS422.IG.xHV_SW, 'MKS422 xHV_SW set to False');
    AssertFalse(This^.fb_MKS422.IG.q_xHV_DIS, 'MKS422 q_xHV_DIS set to True');
    TEST_FINISHED_NAMED('MKS422_Interlock_OK');

    8:
    This^.PG.rPRESS := 1E-1;
    This^.PG.xPRESS_OK := False;
    This^.fb_MKS422(PG:=This^.PG, IG=>);

    11:
    AssertFalse(This^.fb_MKS422.IG.xHV_SW, 'MKS422 xHV_SW set to True');
    AssertTrue(This^.fb_MKS422.IG.q_xHV_DIS, 'MKS422 q_xHV_DIS set to False');
    TEST_FINISHED_NAMED('MKS422_Interlock_Lost');
END_CASE

This^.fb_MKS422(PG:=This^.PG, IG=>);
END_METHOD

METHOD M_SelfProtection
VAR_INPUT
END_VAR
// Switching the Cold cathode backon
TEST('MKS422_Interlock_OK_1');
This^.PG.rPRESS := 1E-4;
This^.PG.xPRESS_OK := True;
fb_MKS422.M_HVE(TRUE);
This^.fb_MKS422(PG:=This^.PG, IG=>);
AssertTrue(This^.fb_MKS422.IG.xHV_SW, 'MKS422 xHV_SW set to False');
AssertFalse(This^.fb_MKS422.IG.q_xHV_DIS, 'MKS422 q_xHV_DIS set to True');
TEST_FINISHED_NAMED('MKS422_Interlock_OK_1');

TEST('MKS422_Self_Protection');
This^.PG.rPRESS := 1E-3;
This^.PG.xPRESS_OK := TRUE;
This^.fb_MKS422(PG:=This^.PG, IG=>);
AssertFalse(This^.fb_MKS422.IG.xHV_SW, 'MKS422 xHV_SW set to True');
AssertTrue(This^.fb_MKS422.IG.q_xHV_DIS, 'MKS422 q_xHV_DIS set to False');
TEST_FINISHED_NAMED('MKS422_Self_Protection');
END_METHOD

END_FUNCTION_BLOCK

// ---- UnitTests/Gauges/FB_GPI_Test.TcPOU
FUNCTION_BLOCK FB_GPI_Test EXTENDS TcUnit.FB_TestSuite
VAR_INPUT
END_VAR
VAR_OUTPUT
END_VAR
VAR
    fb_MKS275: FB_MKS275;
    fb_MKS317: FB_MKS317;
    i_iPRESS_R AT %Q* :INT;
    cycle:INT :=0;
END_VAR

M_INIT();
M_CheckRange();
cycle:=cycle+1;

METHOD M_CheckRange
VAR
    Expected:REAL;
    Actual:REAL;
    eStateExpected: E_PressureState;
    eStateActual: E_PressureState;
END_VAR

TEST('MKS275_Check_Range');
Case cycle of
    4:
    This^.i_iPRESS_R := V_TO_INT(3.674);
    Expected :=5 ;
    eStateExpected := Valid;

    7:
    TEST('MKS275_Range_R2');
    Actual := This^.fb_MKS275.PG.rPRESS;
    eStateActual := This^.fb_MKS275.PG.eState;
    AssertTrue(This^.fb_MKS275.PG.xPRESS_OK, 'MKS275 xPRESS_OK is set to False');
    AssertEquals(eStateExpected,eStateActual,'MKS275 eState Fail');
    AssertEquals_REAL(Expected, Actual,0.1, 'MKS275 rPress Fail');
    TEST_FINISHED_NAMED('MKS275_Range_R2');

    8:
    This^.i_iPRESS_R := V_TO_INT(5.614);
    Expected :=900 ;
    eStateExpected := Valid;


    12:
    TEST('MKS275_Range_R3');
    Actual := This^.fb_MKS275.PG.rPRESS;
    eStateActual := This^.fb_MKS275.PG.eState;
    AssertTrue(This^.fb_MKS275.PG.xPRESS_OK, 'MKS275 xPRESS_OK is set to False');
    AssertEquals(eStateExpected,eStateActual,'MKS275 eState Fail');
    AssertEquals_REAL(Expected, Actual,1, 'MKS275 rPress Fail');
    TEST_FINISHED_NAMED('MKS275_Range_R3');


    13:
    This^.i_iPRESS_R := V_TO_INT(0.3);
    Expected :=-1 ;
    eStateExpected := GaugeDisconnected;

    17:
    TEST('MKS275_Range_Off');
    Actual := This^.fb_MKS275.PG.rPRESS;
    eStateActual := This^.fb_MKS275.PG.eState;
    AssertTrue(This^.fb_MKS275.PG.xPRESS_OK, 'MKS275 xPRESS_OK is set to False');
    AssertEquals(eStateExpected,eStateActual,'MKS275 eState Fail');
    AssertEquals_REAL(Expected, Actual,1, 'MKS275 rPress Fail');
    TEST_FINISHED_NAMED('MKS275_Range_Off');


    18:
    This^.i_iPRESS_R := V_TO_INT(5.66);
    Expected :=-1 ;
    eStateExpected := OoR;

    22:
    TEST('MKS275_Range_OoR');
    Actual := This^.fb_MKS275.PG.rPRESS;
    eStateActual := This^.fb_MKS275.PG.eState;
    AssertTrue(This^.fb_MKS275.PG.xPRESS_OK, 'MKS275 xPRESS_OK is set to False');
    AssertEquals(eStateExpected,eStateActual,'MKS275 eState Fail');
    AssertEquals_REAL(Expected, Actual,1, 'MKS275 rPress Fail');
    TEST_FINISHED_NAMED('MKS275_Range_OoR');
    TEST_FINISHED_NAMED('MKS275_Check_Range');

END_CASE

This^.fb_MKS275(PG=>);
This^.fb_MKS317(PG=>);
END_METHOD

METHOD M_INIT
VAR
    Expected:REAL;
    Actual:REAL;
    eStateExpected: E_PressureState;
    eStateActual: E_PressureState;
END_VAR
// Start the Test
TEST('MKS275_Startup');
//Assign Voltage to FB
This^.i_iPRESS_R := V_TO_INT(0.384);
// Assigne expected result corresponing to the test input
Expected :=0.001 ;
eStateExpected := Valid;
//Instantiate the function block
This^.fb_MKS275(PG=>);
// Wait for few cycles
IF( cycle = 3) THEN
    // Check the results
    Actual := This^.fb_MKS275.PG.rPRESS;
    eStateActual := This^.fb_MKS275.PG.eState;
    AssertTrue(This^.fb_MKS275.PG.xPRESS_OK, 'MKS275 xPRESS_OK is set to False');
    AssertEquals(eStateExpected,eStateActual,'MKS275 eState Fail');
    AssertEquals_REAL(Expected, Actual,0.0001, 'MKS275 rPress Fail');
    TEST_FINISHED_NAMED('MKS275_Startup');
END_IF
END_METHOD

END_FUNCTION_BLOCK

// ---- UnitTests/Pumps/FB_PIP_Test.TcPOU
FUNCTION_BLOCK FB_PIP_Test EXTENDS TcUnit.FB_TestSuite
VAR_INPUT
END_VAR
VAR_OUTPUT
END_VAR
VAR
    PG : ST_VG;
    fb_PIP_GAMMA: FB_PIP_GAMMA;
END_VAR

M_INIT();
M_Interlock();
M_AutoStart();

METHOD M_AutoStart
VAR_INPUT
END_VAR
TEST('PIP_Auto_Restart');
This^.PG.rPRESS := 1E-6;
This^.PG.xPRESS_OK := TRUE;
This^.fb_PIP_GAMMA(i_stGauge:=PG, stPump=>, q_IG=>);
AssertTrue(This^.fb_PIP_GAMMA.stPump.q_xHVEna_DO, 'PIP HVEna_DO set to false');
TEST_FINISHED_NAMED('PIP_Auto_Restart');
END_METHOD

METHOD M_Check_State
VAR_INPUT
END_VAR
END_METHOD

METHOD M_INIT
VAR_INPUT
END_VAR
TEST('PIP_Startup');
This^.PG.rPRESS := 1E-1;
This^.PG.xPRESS_OK := TRUE;
This^.fb_PIP_GAMMA(i_stGauge:=PG, stPump=>, q_IG=>);
AssertFalse(This^.fb_PIP_GAMMA.stPump.xHVEna_SW, 'PIP xHVEna_SW set to True');
AssertFalse(This^.fb_PIP_GAMMA.stPump.q_xHVEna_DO, 'PIP HVEna_DO set to True');
TEST_FINISHED_NAMED('PIP_Startup');
END_METHOD

METHOD M_Interlock
VAR_INPUT
END_VAR
TEST('PIP_Interlock_Active');
This^.PG.rPRESS := 1E-1;
This^.PG.xPRESS_OK := True;
This^.fb_PIP_GAMMA.M_Run(TRUE);
This^.fb_PIP_GAMMA(i_stGauge:=PG, stPump=>, q_IG=>);
AssertFalse(This^.fb_PIP_GAMMA.stPump.xHVEna_SW, 'PIP xHVEna_SW set to True');
AssertFalse(This^.fb_PIP_GAMMA.stPump.q_xHVEna_DO, 'PIP HVEna_DO set to True');
TEST_FINISHED_NAMED('PIP_Interlock_Active');

TEST('PIP_Interlock_OK');
This^.PG.rPRESS := 1E-9;
This^.PG.xPRESS_OK := True;
This^.fb_PIP_GAMMA.M_Run(TRUE);
This^.fb_PIP_GAMMA(i_stGauge:=PG, stPump=>, q_IG=>);
AssertTrue(This^.fb_PIP_GAMMA.stPump.xHVEna_SW, 'PIP xHVEna_SW set to False');
AssertTrue(This^.fb_PIP_GAMMA.stPump.q_xHVEna_DO, 'PIP HVEna_DO set to False');
TEST_FINISHED_NAMED('PIP_Interlock_OK');

TEST('PIP_Interlock_Lost');
This^.PG.rPRESS := 1E-9;
This^.PG.xPRESS_OK := False;
This^.fb_PIP_GAMMA(i_stGauge:=PG, stPump=>, q_IG=>);
AssertFalse(This^.fb_PIP_GAMMA.stPump.xHVEna_SW, 'PIP xHVEna_SW set to True');
AssertFalse(This^.fb_PIP_GAMMA.stPump.q_xHVEna_DO, 'PIP HVEna_DO set to True');
TEST_FINISHED_NAMED('PIP_Interlock_Lost');
END_METHOD

END_FUNCTION_BLOCK

// ---- UnitTests/Pumps/FB_PTM_Test.TcPOU
FUNCTION_BLOCK FB_PTM_Test EXTENDS TcUnit.FB_TestSuite
VAR_INPUT
END_VAR
VAR_OUTPUT
END_VAR
VAR
    fb_TwisTorr: FB_PTM_TwisTorr;
    fb_PTM_Ebara_010M:FB_PTM_Ebara_010M;

    cycle:INT :=0;
    (*IO*)
    q_iSpeedSet AT %I* :INT;
    i_diCurSpd AT %Q* :INT;

    i_iRawSpeed AT %Q* : INT; // Link to Analog input
    i_iTempMon AT %Q* : INT; // Link to Analog input -- input Voltage according to the pump temprature 0->5V 0->100C
    i_iCurrentMon AT %Q* : INT; //Link to Analog -- input Voltage to the output current of motor 0->5V 0->10A

END_VAR

M_INIT();
M_Interlock();
M_PTM_EBARA();
cycle:=cycle+1;

METHOD M_INIT : BOOL
VAR_INPUT
END_VAR
TEST('PTM_Twistorr_Startup');
fb_TwisTorr(i_xExtILKOk:= TRUE , iq_stPtm=> );
IF( cycle = 3) THEN
    AssertFalse(fb_TwisTorr.iq_stPtm.xRunSW ,'PTM Twistorr xRunSW is set to true');
    AssertFalse(fb_TwisTorr.iq_stPtm.q_RunDO ,'PTM Twistorr q_RunDO is set to true');
    TEST_FINISHED_NAMED('PTM_Twistorr_Startup');
END_IF


TEST('PTM_Ebara011M_Startup');
fb_PTM_Ebara_010M(i_xExtILKOk:= TRUE , iq_stPtm=> );
IF( cycle = 3) THEN
    AssertFalse(fb_PTM_Ebara_010M.iq_stPtm.xRunSW ,'PTM Ebara011M xRunSW is set to true');
    AssertFalse(fb_PTM_Ebara_010M.iq_stPtm.q_RunDO ,'PTM Ebara011M q_RunDO is set to true');
    AssertFalse(fb_PTM_Ebara_010M.iq_stPtm.q_xProtection ,'PTM Ebara011M q_xProtection is set to True');
    TEST_FINISHED_NAMED('PTM_Ebara011M_Startup');
END_IF
END_METHOD

METHOD M_Interlock
VAR_INPUT
END_VAR
TEST('PTM_Twistorr_Interlock_Active');
fb_TwisTorr.M_Run(TRUE);
fb_TwisTorr(i_xExtILKOk:= FALSE , iq_stPtm=> );
IF( cycle = 3) THEN
    AssertFalse(fb_TwisTorr.iq_stPtm.xRunSW ,'PTM Twistorr xRunSW is set to true');
    AssertFalse(fb_TwisTorr.iq_stPtm.q_RunDO ,'PTM Twistorr q_RunDO is set to true');
    TEST_FINISHED_NAMED('PTM_Twistorr_Interlock_Active');
END_IF

TEST('PTM_Twistorr_Interlock_OK');
fb_TwisTorr.M_Run(TRUE);
fb_TwisTorr(i_xExtILKOk:= TRUE , iq_stPtm=> );
IF( cycle = 3) THEN
    AssertTrue(fb_TwisTorr.iq_stPtm.xRunSW ,'PTM Twistorr xRunSW is set to False');
    AssertTrue(fb_TwisTorr.iq_stPtm.q_RunDO ,'PTM Twistorr q_RunDO is set to False');
    TEST_FINISHED_NAMED('PTM_Twistorr_Interlock_OK');
END_IF

TEST('PTM_Twistorr_Interlock_Lost');
fb_TwisTorr(i_xExtILKOk:= FALSE , iq_stPtm=> );
IF( cycle = 3) THEN
    AssertFalse(fb_TwisTorr.iq_stPtm.xRunSW ,'PTM Twistorr xRunSW is set to true');
    AssertFalse(fb_TwisTorr.iq_stPtm.q_RunDO ,'PTM Twistorr q_RunDO is set to true');
    TEST_FINISHED_NAMED('PTM_Twistorr_Interlock_Lost');
END_IF
END_METHOD

METHOD M_PTM_EBARA
VAR
    Expected:REAL;
    Actual:REAL;
    diExpected:DINT;
    diActual: DINT;
END_VAR
TEST('PTM_EBARA_AI');
This^.i_iRawSpeed := v_to_int(5);
This^.i_iTempMon := v_to_int(2.5);
THIS^.i_iCurrentMon := v_to_int(2.5);
//THIS^.q_iSpeedSet := 560;

fb_PTM_Ebara_010M(
    i_xExtILKOk:= TRUE ,
    i_rMaxBackingPressure:= 1,
    iq_stPTM=> );


IF( cycle = 10) THEN
    Expected := 5;
    Actual := (fb_PTM_Ebara_010M.iq_stPTM.i_rCurrentMon);
    AssertEquals_REAL(Expected, Actual,0.1, 'PTM EBARA010 i_iCurrentMon Fail');
    Expected := 50;
    Actual := (fb_PTM_Ebara_010M.iq_stPTM.i_rTempMon);
    AssertEquals_REAL(Expected, Actual,0.1, 'PTM EBARA010 i_iTempMon Fail');
    diExpected := 0;
    diActual := fb_PTM_Ebara_010M.iq_stPTM.q_iSpeedSet;
    AssertEquals(diExpected, diActual, 'PTM EBARA010 q_iSpeedSet Fail');
    diExpected := 560;
    diActual :=  fb_PTM_Ebara_010M.iq_stPTM.i_diCurSpd;
    AssertEquals(diExpected, diActual, 'PTM EBARA010 i_diCurSpd Fail');
    TEST_FINISHED_NAMED('PTM_EBARA_AI');


End_IF;
END_METHOD

END_FUNCTION_BLOCK

// ---- UnitTests/Valves/FB_VGC_Test.TcPOU
FUNCTION_BLOCK FB_VGC_Test EXTENDS TcUnit.FB_TestSuite
VAR_INPUT
END_VAR
VAR_OUTPUT
END_VAR
VAR
    VGC: FB_VGC;
    US_IG : ST_VG;
    DS_IG : ST_VG;
    io_fbFFHWO    :    FB_HardwareFFOutput;
    TotalTests : INT:=0;
    ex               : __SYSTEM.ExceptionCode;
END_VAR

M_INIT();
M_Interlock();

METHOD M_Check_State
VAR_INPUT
END_VAR
END_METHOD

METHOD M_INIT : BOOL
VAR//_INPUT

END_VAR
TEST('VGC_Startup');
This^.US_IG.rPRESS := 1E-9;
This^.US_IG.xPRESS_OK := TRUE;
This^.US_IG.xAT_VAC := TRUE;

This^.DS_IG.rPRESS := 1E-9;
This^.DS_IG.xPRESS_OK := TRUE;

(*This^.VGC(
    i_stUSG:= This^.US_IG,
    i_stDSG:= This^.DS_IG ,
    i_xDis_DPIlk:= FALSE,
    i_xEPS_OK:= TRUE ,
    //i_xPMPS_OK:= TRUE,
    i_xExt_OK:= TRUE,
    i_xOverrideMode:= ,
    i_xReset:= ,
    iq_stValve=> ,
    xMPS_OK=> ,
    io_fbFFHWO:= This^.io_fbFFHWO,
    fbArbiter:=g_fbArbiter);
*)
AssertFalse(This^.VGC.iq_stValve.pv_xOPN_SW,'VGC pv_xOPN_SW is set to true');
AssertFalse(VGC.iq_stValve.q_xOPN_DO,'VGC q_xOPN_DO is set to true');
TEST_FINISHED_NAMED('VGC_Startup');
END_METHOD

METHOD M_Interlock : BOOL
VAR//_INPUT

END_VAR
// Test interlock is active and attempting to open valve
TEST('VGC_Interlock_Active');
This^.US_IG.xPRESS_OK := FALSE;
This^.DS_IG.xPRESS_OK := FALSE;
VGC.M_Set_OPN_SW(TRUE);
// run the function block one more time
(*VGC(
    i_stUSG:= US_IG,
    i_stDSG:= DS_IG ,
    i_xDis_DPIlk:= FALSE,
    i_xEPS_OK:= TRUE ,
    i_xPMPS_OK:= TRUE ,
    i_xExt_OK:= TRUE,
    i_xOverrideMode:= ,
    i_xReset:= ,
    iq_stValve=> ,
    xMPS_OK=> ,
    io_fbFFHWO:= io_fbFFHWO);*)
AssertFalse(VGC.iq_stValve.pv_xOPN_SW,'VGC pv_xOPN_SW is set to true');
AssertFalse(VGC.iq_stValve.q_xOPN_DO,'VGC q_xOPN_DO is set to true');
TEST_FINISHED_NAMED('VGC_Interlock_Active');
// Test interlock is not active and attempting to open valve
TEST('VGC_Interlock_OK');
This^.US_IG.xPRESS_OK := TRUE;
This^.DS_IG.xPRESS_OK := TRUE;
VGC.M_Set_OPN_SW(TRUE);
// run the function block one more time
(*VGC(
    i_stUSG:= US_IG,
    i_stDSG:= DS_IG ,
    i_xDis_DPIlk:= FALSE,
    i_xEPS_OK:= ,
    i_xPMPS_OK:= ,
    i_xExt_OK:= ,
    i_xOverrideMode:= ,
    i_xReset:= ,
    iq_stValve=> ,
    xMPS_OK=> ,
    io_fbFFHWO:= io_fbFFHWO);*)
AssertTrue(VGC.iq_stValve.pv_xOPN_SW,'VGC pv_xOPN_SW is set to false');
AssertTrue(VGC.iq_stValve.q_xOPN_DO,'VGC q_xOPN_DO is set to false');
TEST_FINISHED_NAMED('VGC_Interlock_OK');
// Test interlock ok lost while valve is open
TEST('VGC_Interlock_Lost');
This^.US_IG.xPRESS_OK := False;
This^.DS_IG.xPRESS_OK := TRUE;
// run the function block one more time
(*VGC(
    i_stUSG:= US_IG,
    i_stDSG:= DS_IG ,
    i_xDis_DPIlk:= FALSE,
    i_xEPS_OK:= ,
    i_xPMPS_OK:= ,
    i_xExt_OK:= ,
    i_xOverrideMode:= ,
    i_xReset:= ,
    iq_stValve=> ,
    xMPS_OK=> ,
    io_fbFFHWO:= io_fbFFHWO);*)
AssertFalse(VGC.iq_stValve.pv_xOPN_SW,'VGC pv_xOPN_SW is set to true');
AssertFalse(VGC.iq_stValve.q_xOPN_DO,'VGC q_xOPN_DO is set to true');
TEST_FINISHED_NAMED('VGC_Interlock_Lost');
END_METHOD

END_FUNCTION_BLOCK

// ---- UnitTests/Valves/FB_VRC_Test.TcPOU
FUNCTION_BLOCK FB_VRC_Test EXTENDS TcUnit.FB_TestSuite
VAR_INPUT
END_VAR
VAR_OUTPUT
END_VAR
VAR
    VRC: FB_VRC;
    ex               : __SYSTEM.ExceptionCode;
END_VAR

M_INIT();
M_Interlock();

METHOD M_Check_State
VAR_INPUT
END_VAR
END_METHOD

METHOD M_INIT : BOOL
VAR//_INPUT


    Interlock_OK :BOOL := TRUE;

    ex: INT;
END_VAR
TEST('VRC_Startup');
//__TRY
VRC(i_xExtILK_OK:= Interlock_OK, i_xOverrideMode:= , iq_stValve=> );
AssertFalse(VRC.iq_stValve.q_xOPN_DO,'VRC q_xOPN_DO is set to true');
AssertFalse(VRC.iq_stValve.pv_xOPN_SW,'VRC pv_xOPN_SW is set to true');
//__CATCH(ex)
//__FINALLY
TEST_FINISHED_NAMED('VRC_Startup');
//__ENDTRY
END_METHOD

METHOD M_Interlock
VAR
    US_IG : ST_VG;
    DS_IG : ST_VG;

    VRC: FB_VRC;
END_VAR
TEST('VRC_Interlock_Active');
VRC.M_Set_OPN_SW (TRUE);
VRC(i_xExtILK_OK:= FALSE, i_xOverrideMode:= , iq_stValve=> );
AssertFalse(VRC.iq_stValve.pv_xOPN_SW,'VRC open_SW is set to true');
AssertFalse(VRC.iq_stValve.q_xOPN_DO,'VRC open DO is set to true');
TEST_FINISHED_NAMED('VRC_Interlock_Active');

TEST('VRC_Interlock_OK');
VRC.M_Set_OPN_SW (TRUE);
VRC(i_xExtILK_OK:= TRUE, i_xOverrideMode:= , iq_stValve=> );
AssertTrue(VRC.iq_stValve.pv_xOPN_SW,'VRC open_SW is set to FALSE');
AssertTrue(VRC.iq_stValve.q_xOPN_DO,'VRC open DO is set to FALSE');
TEST_FINISHED_NAMED('VRC_Interlock_OK');

TEST('VRC_Interlock_Lost');
VRC(i_xExtILK_OK:= FALSE, i_xOverrideMode:= , iq_stValve=> );
AssertFalse(VRC.iq_stValve.pv_xOPN_SW,'VRC open_SW is set to true');
AssertFalse(VRC.iq_stValve.q_xOPN_DO,'VRC open DO is set to true');
TEST_FINISHED_NAMED('VRC_Interlock_Lost');
END_METHOD

END_FUNCTION_BLOCK
